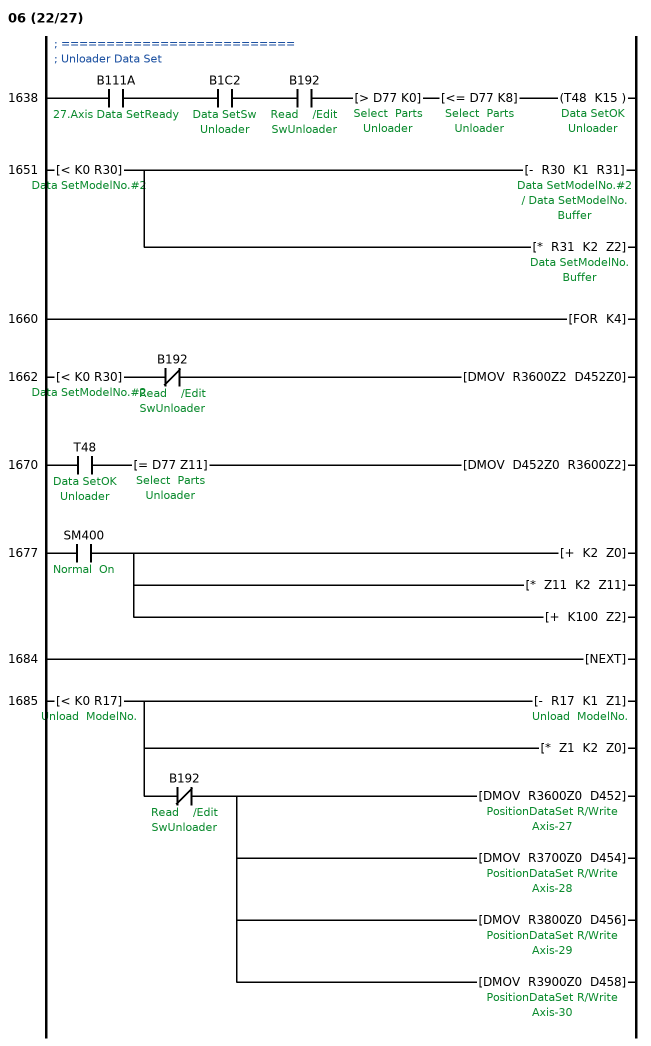
; ==========================
; Unloader Data Set
1638  LD      B111A  ; 27.Axis Data SetReady
      AND     B1C2  ; Data SetSw      Unloader
      AND     B192  ; Read    /Edit SwUnloader
      AND>    D77 K0  ; Select  Parts   Unloader
      AND<=   D77 K8  ; Select  Parts   Unloader
      OUT     T48 K15  ; Data SetOK      Unloader
1651  LD<     K0 R30  ; Data SetModelNo.#2
      -       R30 K1 R31
      *       R31 K2 Z2
1660  FOR     K4
1662  LD<     K0 R30  ; Data SetModelNo.#2
      ANI     B192  ; Read    /Edit SwUnloader
      DMOV    R3600Z2 D452Z0
1670  LD      T48  ; Data SetOK      Unloader
      AND=    D77 Z11  ; Select  Parts   Unloader
      DMOV    D452Z0 R3600Z2
1677  LD      SM400  ; Normal  On
      +       K2 Z0
      *       Z11 K2 Z11
      +       K100 Z2
1684  NEXT
1685  LD<     K0 R17  ; Unload  ModelNo.
      -       R17 K1 Z1
      *       Z1 K2 Z0
      ANI     B192  ; Read    /Edit SwUnloader
      DMOV    R3600Z0 D452  ; PositionDataSet R/Write Axis-27
      DMOV    R3700Z0 D454  ; PositionDataSet R/Write Axis-28
      DMOV    R3800Z0 D456  ; PositionDataSet R/Write Axis-29
      DMOV    R3900Z0 D458  ; PositionDataSet R/Write Axis-30
      P1
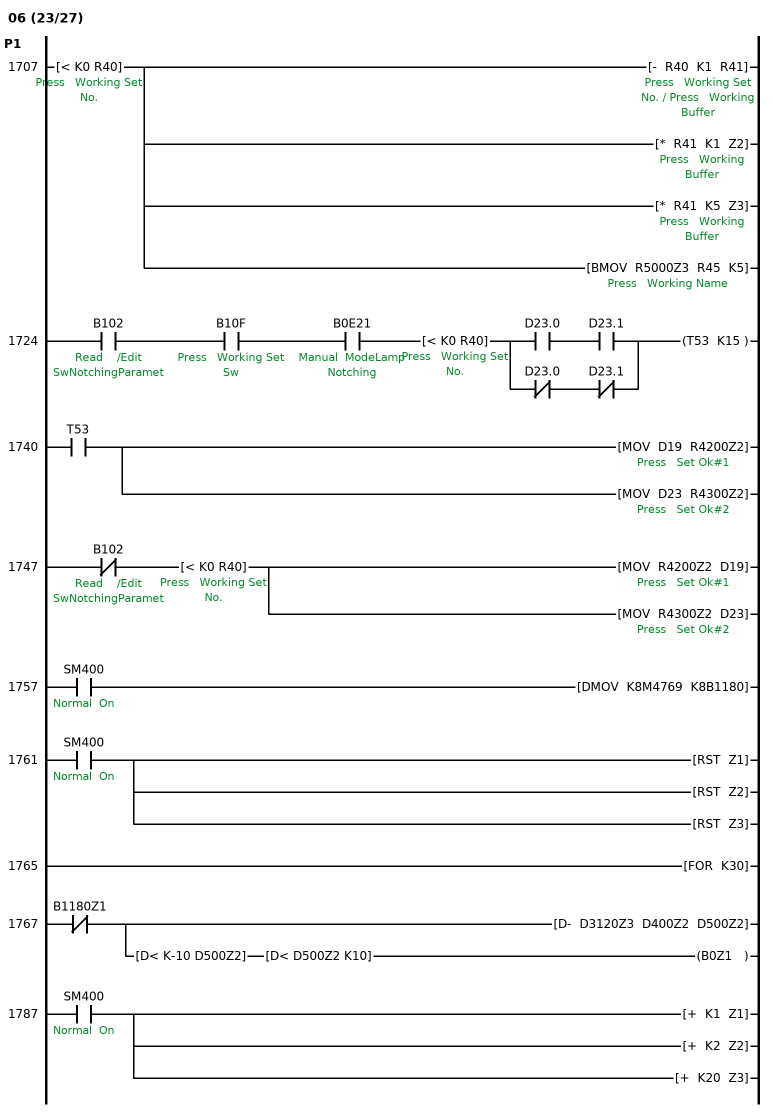
1707  LD<     K0 R40  ; Press   Working Set No.
      -       R40 K1 R41  ; Press   Working Buffer
      *       R41 K1 Z2
      *       R41 K5 Z3
      BMOV    R5000Z3 R45 K5  ; Press   Working Name
1724  LD      B102  ; Read    /Edit SwNotchingParamet
      AND     B10F  ; Press   Working Set Sw
      AND     B0E21  ; Manual  ModeLampNotching
      AND<    K0 R40  ; Press   Working Set No.
      LD      D23.0
      AND     D23.1
      LDI     D23.0
      ANI     D23.1
      ORB
      ANB
      OUT     T53 K15
1740  LD      T53
      MOV     D19 R4200Z2
      MOV     D23 R4300Z2
1747  LDI     B102  ; Read    /Edit SwNotchingParamet
      AND<    K0 R40  ; Press   Working Set No.
      MOV     R4200Z2 D19
      MOV     R4300Z2 D23
1757  LD      SM400  ; Normal  On
      DMOV    K8M4769 K8B1180  ; 1.Axis  Busy
1761  LD      SM400  ; Normal  On
      RST     Z1
      RST     Z2
      RST     Z3
1765  FOR     K30
1767  LDI     B1180Z1
      D-      D3120Z3 D400Z2 D500Z2
      ANDD<   K-10 D500Z2
      ANDD<   D500Z2 K10
      OUT     B0Z1
1787  LD      SM400  ; Normal  On
      +       K1 Z1
      +       K2 Z2
      +       K20 Z3
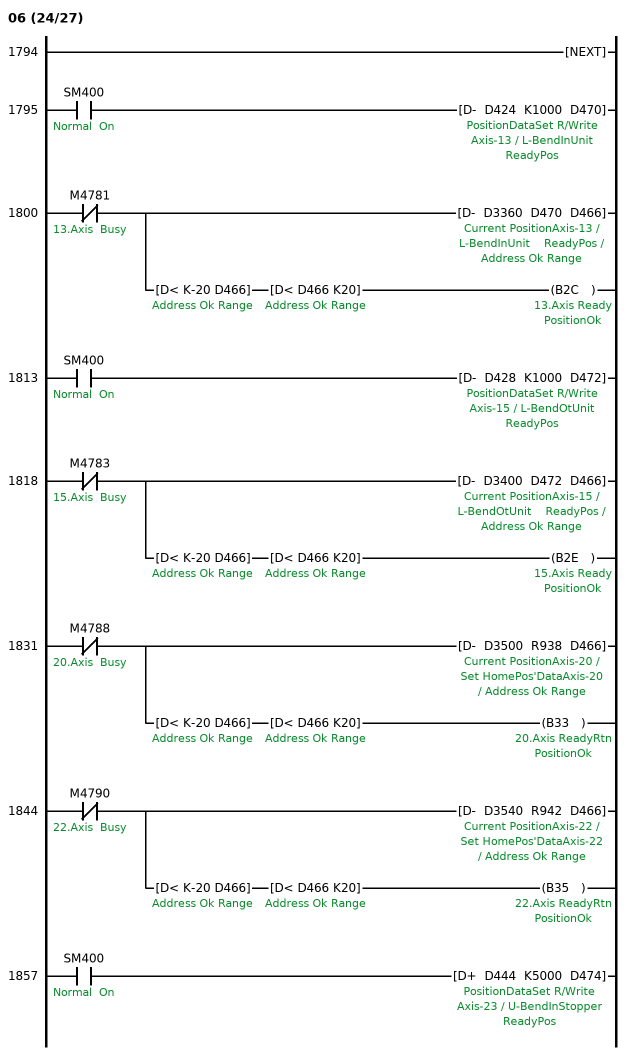
1794  NEXT
1795  LD      SM400  ; Normal  On
      D-      D424 K1000 D470  ; L-BendInUnit    ReadyPos
1800  LDI     M4781  ; 13.Axis  Busy
      D-      D3360 D470 D466  ; Current PositionAxis-13 / Address Ok Range
      ANDD<   K-20 D466  ; Address Ok Range
      ANDD<   D466 K20  ; Address Ok Range
      OUT     B2C  ; 13.Axis Ready   PositionOk
1813  LD      SM400  ; Normal  On
      D-      D428 K1000 D472  ; L-BendOtUnit    ReadyPos
1818  LDI     M4783  ; 15.Axis  Busy
      D-      D3400 D472 D466  ; Current PositionAxis-15
      ANDD<   K-20 D466  ; Address Ok Range
      ANDD<   D466 K20  ; Address Ok Range
      OUT     B2E  ; 15.Axis Ready   PositionOk
1831  LDI     M4788  ; 20.Axis  Busy
      D-      D3500 R938 D466  ; Current PositionAxis-20 / Set HomePos'DataAxis-20
      ANDD<   K-20 D466  ; Address Ok Range
      ANDD<   D466 K20  ; Address Ok Range
      OUT     B33  ; 20.Axis ReadyRtnPositionOk
1844  LDI     M4790  ; 22.Axis  Busy
      D-      D3540 R942 D466  ; Current PositionAxis-22 / Set HomePos'DataAxis-22
      ANDD<   K-20 D466  ; Address Ok Range
      ANDD<   D466 K20  ; Address Ok Range
      OUT     B35  ; 22.Axis ReadyRtnPositionOk
1857  LD      SM400  ; Normal  On
      D+      D444 K5000 D474  ; U-BendInStopper ReadyPos
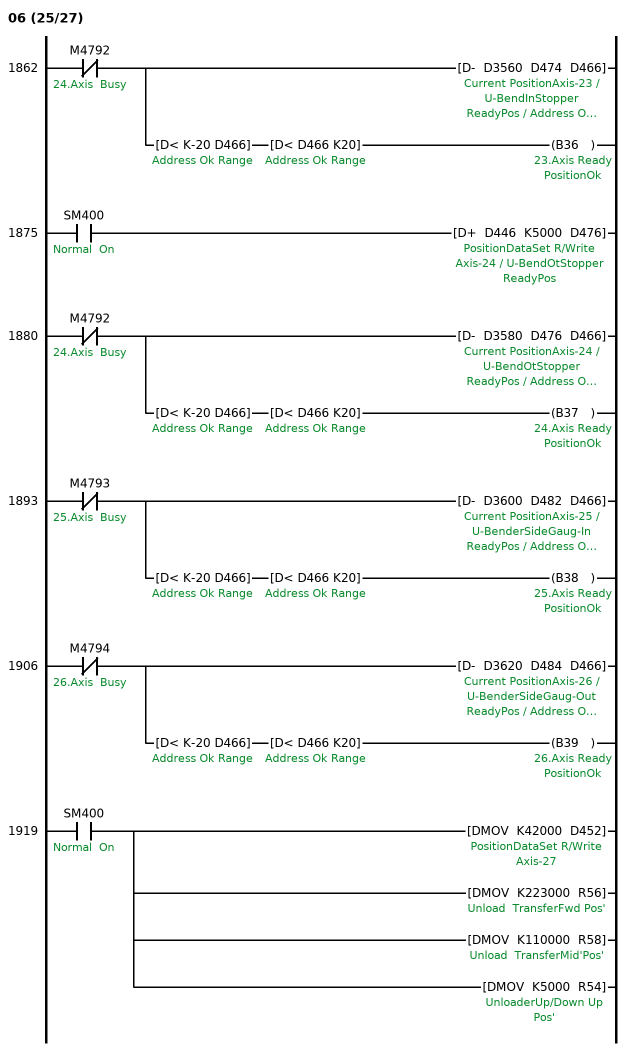
1862  LDI     M4792  ; 24.Axis  Busy
      D-      D3560 D474 D466  ; Current PositionAxis-23
      ANDD<   K-20 D466  ; Address Ok Range
      ANDD<   D466 K20  ; Address Ok Range
      OUT     B36  ; 23.Axis Ready   PositionOk
1875  LD      SM400  ; Normal  On
      D+      D446 K5000 D476  ; U-BendOtStopper ReadyPos
1880  LDI     M4792  ; 24.Axis  Busy
      D-      D3580 D476 D466  ; Current PositionAxis-24
      ANDD<   K-20 D466  ; Address Ok Range
      ANDD<   D466 K20  ; Address Ok Range
      OUT     B37  ; 24.Axis Ready   PositionOk
1893  LDI     M4793  ; 25.Axis  Busy
      D-      D3600 D482 D466  ; Current PositionAxis-25 / U-BenderSideGaug-In     ReadyPos
      ANDD<   K-20 D466  ; Address Ok Range
      ANDD<   D466 K20  ; Address Ok Range
      OUT     B38  ; 25.Axis Ready   PositionOk
1906  LDI     M4794  ; 26.Axis  Busy
      D-      D3620 D484 D466  ; Current PositionAxis-26 / U-BenderSideGaug-Out    ReadyPos
      ANDD<   K-20 D466  ; Address Ok Range
      ANDD<   D466 K20  ; Address Ok Range
      OUT     B39  ; 26.Axis Ready   PositionOk
1919  LD      SM400  ; Normal  On
      DMOV    K42000 D452
      DMOV    K223000 R56  ; Unload  TransferFwd Pos'
      DMOV    K110000 R58  ; Unload  TransferMid'Pos'
      DMOV    K5000 R54  ; UnloaderUp/Down Up Pos'
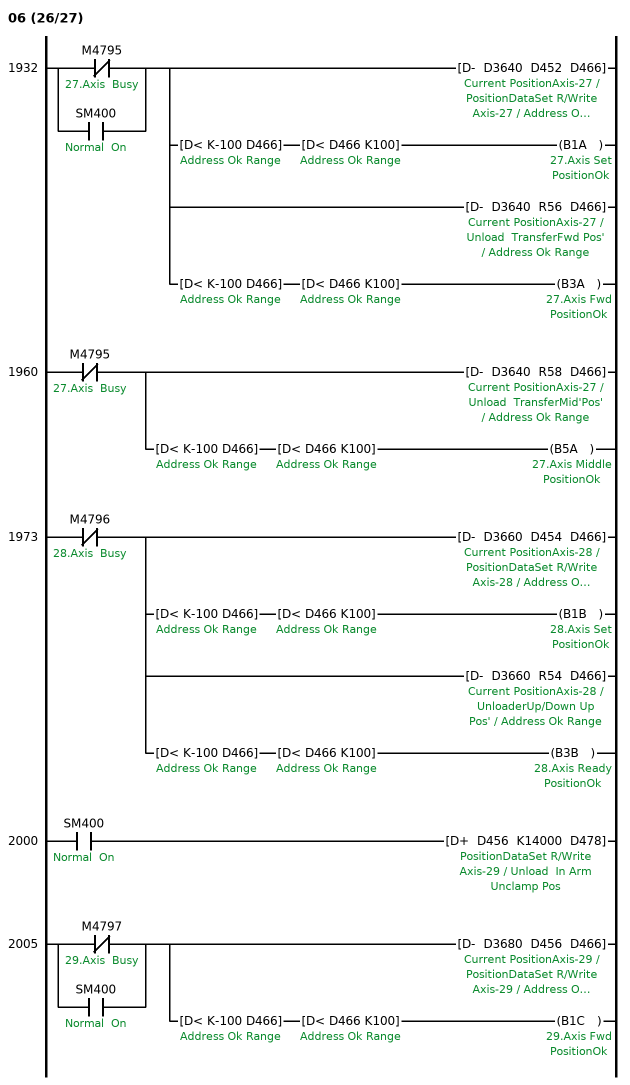
1932  LDI     M4795  ; 27.Axis  Busy
      OR      SM400  ; Normal  On
      D-      D3640 D452 D466  ; Current PositionAxis-27
      MPS
      ANDD<   K-100 D466  ; Address Ok Range
      ANDD<   D466 K100  ; Address Ok Range
      OUT     B1A  ; 27.Axis Set     PositionOk
      MPP
      D-      D3640 R56 D466
      ANDD<   K-100 D466  ; Address Ok Range
      ANDD<   D466 K100  ; Address Ok Range
      OUT     B3A  ; 27.Axis Fwd     PositionOk
1960  LDI     M4795  ; 27.Axis  Busy
      D-      D3640 R58 D466
      ANDD<   K-100 D466  ; Address Ok Range
      ANDD<   D466 K100  ; Address Ok Range
      OUT     B5A  ; 27.Axis Middle  PositionOk
1973  LDI     M4796  ; 28.Axis  Busy
      D-      D3660 D454 D466  ; Current PositionAxis-28
      MPS
      ANDD<   K-100 D466  ; Address Ok Range
      ANDD<   D466 K100  ; Address Ok Range
      OUT     B1B  ; 28.Axis Set     PositionOk
      MPP
      D-      D3660 R54 D466
      ANDD<   K-100 D466  ; Address Ok Range
      ANDD<   D466 K100  ; Address Ok Range
      OUT     B3B  ; 28.Axis Ready   PositionOk
2000  LD      SM400  ; Normal  On
      D+      D456 K14000 D478  ; Unload  In Arm  Unclamp Pos
2005  LDI     M4797  ; 29.Axis  Busy
      OR      SM400  ; Normal  On
      D-      D3680 D456 D466  ; Current PositionAxis-29
      ANDD<   K-100 D466  ; Address Ok Range
      ANDD<   D466 K100  ; Address Ok Range
      OUT     B1C  ; 29.Axis Fwd     PositionOk
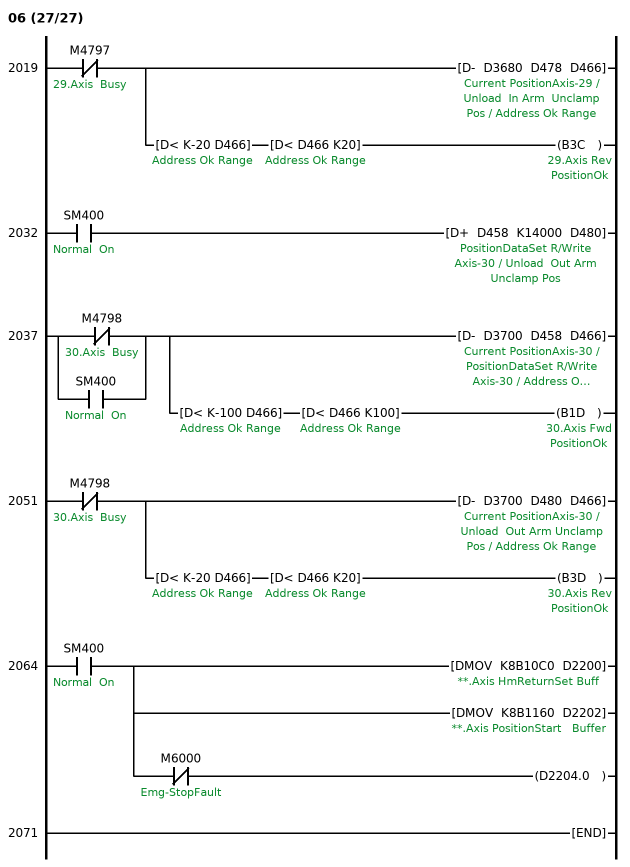
2019  LDI     M4797  ; 29.Axis  Busy
      D-      D3680 D478 D466
      ANDD<   K-20 D466  ; Address Ok Range
      ANDD<   D466 K20  ; Address Ok Range
      OUT     B3C  ; 29.Axis Rev     PositionOk
2032  LD      SM400  ; Normal  On
      D+      D458 K14000 D480  ; Unload  Out Arm Unclamp Pos
2037  LDI     M4798  ; 30.Axis  Busy
      OR      SM400  ; Normal  On
      D-      D3700 D458 D466  ; Current PositionAxis-30
      ANDD<   K-100 D466  ; Address Ok Range
      ANDD<   D466 K100  ; Address Ok Range
      OUT     B1D  ; 30.Axis Fwd     PositionOk
2051  LDI     M4798  ; 30.Axis  Busy
      D-      D3700 D480 D466
      ANDD<   K-20 D466  ; Address Ok Range
      ANDD<   D466 K20  ; Address Ok Range
      OUT     B3D  ; 30.Axis Rev     PositionOk
2064  LD      SM400  ; Normal  On
      DMOV    K8B10C0 D2200  ; 01.Axis HmReturnSet / **.Axis HmReturnSet Buff
      DMOV    K8B1160 D2202  ; 01.Axis PositionStart / **.Axis PositionStart   Buffer
      ANI     M6000  ; Emg-StopFault
      OUT     D2204.0
2071  END
END_PROGRAM

PROGRAM 10  // #1 Conveyor Part
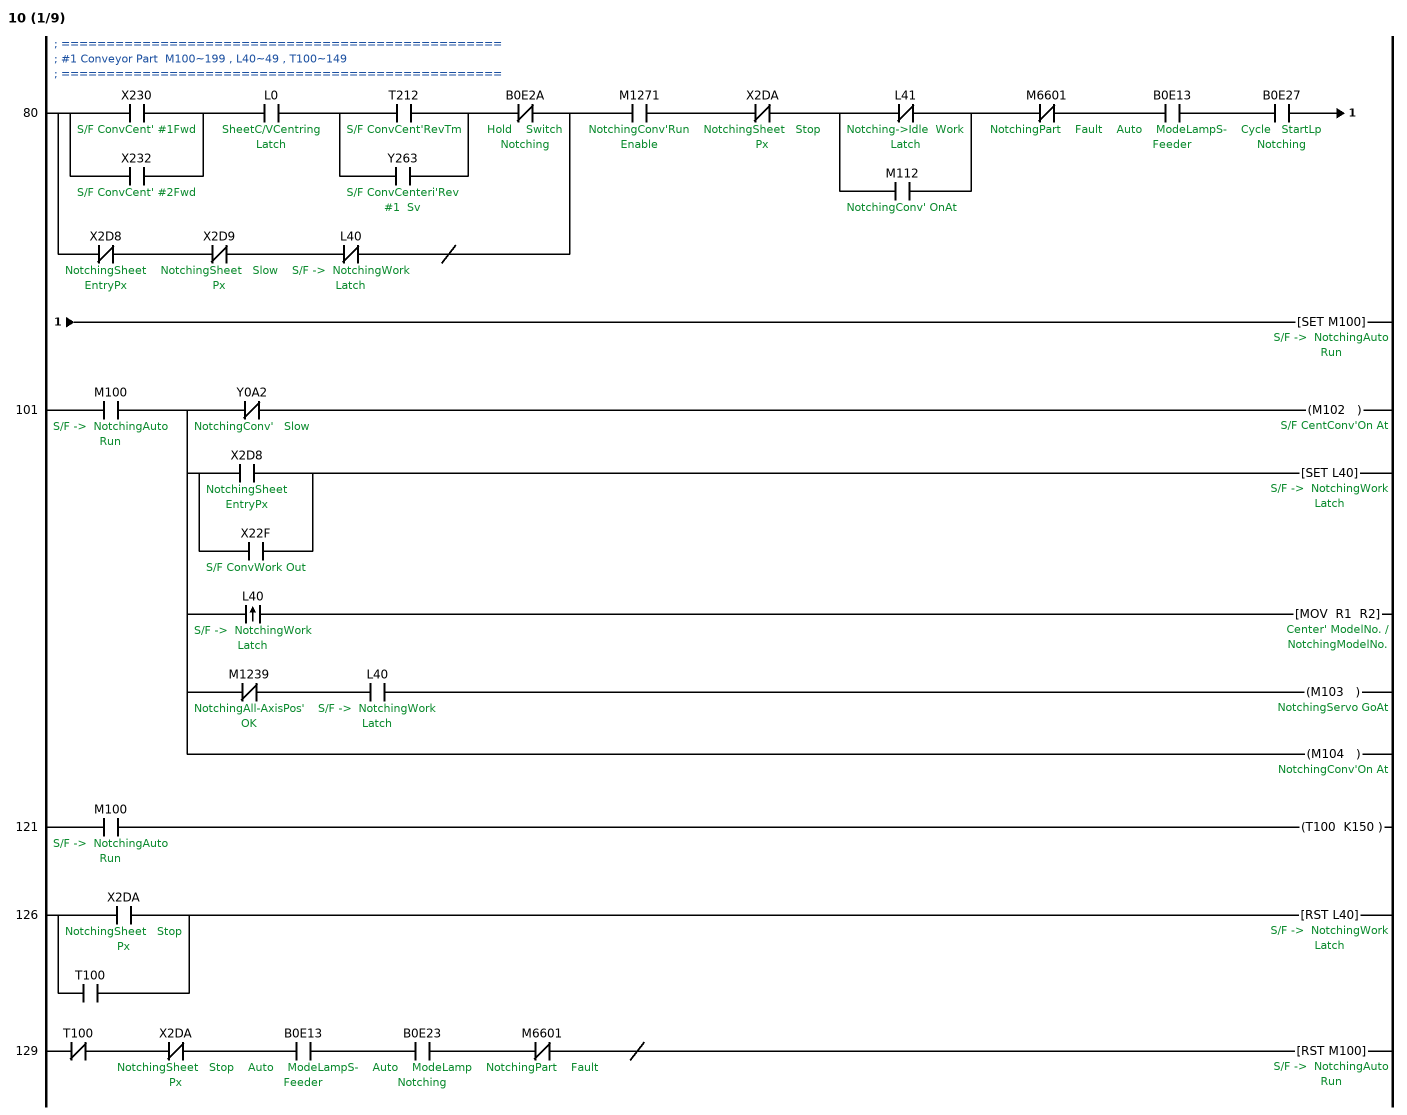
; =================================================
; #1 Conveyor Part  M100~199 , L40~49 , T100~149
; =================================================
80    LD      X230  ; S/F ConvCent' #1Fwd
      OR      X232  ; S/F ConvCent' #2Fwd
      AND     L0  ; SheetC/VCentringLatch
      LD      T212  ; S/F ConvCent'RevTm
      OR      Y263  ; S/F ConvCenteri'Rev #1  Sv
      ANB
      ANI     B0E2A  ; Hold    Switch  Notching
      LDI     X2D8  ; NotchingSheet   EntryPx
      ANI     X2D9  ; NotchingSheet   Slow Px
      ANI     L40  ; S/F ->  NotchingWork    Latch
      INV
      ORB
      AND     M1271  ; NotchingConv'RunEnable
      ANI     X2DA  ; NotchingSheet   Stop Px
      LDI     L41  ; Notching->Idle  Work    Latch
      OR      M112  ; NotchingConv' OnAt
      ANB
      ANI     M6601  ; NotchingPart    Fault
      AND     B0E13  ; Auto    ModeLampS-Feeder
      AND     B0E27  ; Cycle   StartLp Notching
      SET     M100  ; S/F ->  NotchingAuto Run
101   LD      M100  ; S/F ->  NotchingAuto Run
      MPS
      ANI     Y0A2  ; NotchingConv'   Slow
      OUT     M102  ; S/F CentConv'On At
      MRD
      LD      X2D8  ; NotchingSheet   EntryPx
      OR      X22F  ; S/F ConvWork Out
      ANB
      SET     L40  ; S/F ->  NotchingWork    Latch
      MRD
      ANDP    L40  ; S/F ->  NotchingWork    Latch
      MOV     R1 R2  ; Center' ModelNo. / NotchingModelNo.
      MRD
      ANI     M1239  ; NotchingAll-AxisPos' OK
      AND     L40  ; S/F ->  NotchingWork    Latch
      OUT     M103  ; NotchingServo GoAt
      MPP
      OUT     M104  ; NotchingConv'On At
121   LD      M100  ; S/F ->  NotchingAuto Run
      OUT     T100 K150
126   LD      X2DA  ; NotchingSheet   Stop Px
      OR      T100
      RST     L40  ; S/F ->  NotchingWork    Latch
129   LDI     T100
      ANI     X2DA  ; NotchingSheet   Stop Px
      AND     B0E13  ; Auto    ModeLampS-Feeder
      AND     B0E23  ; Auto    ModeLampNotching
      ANI     M6601  ; NotchingPart    Fault
      INV
      RST     M100  ; S/F ->  NotchingAuto Run
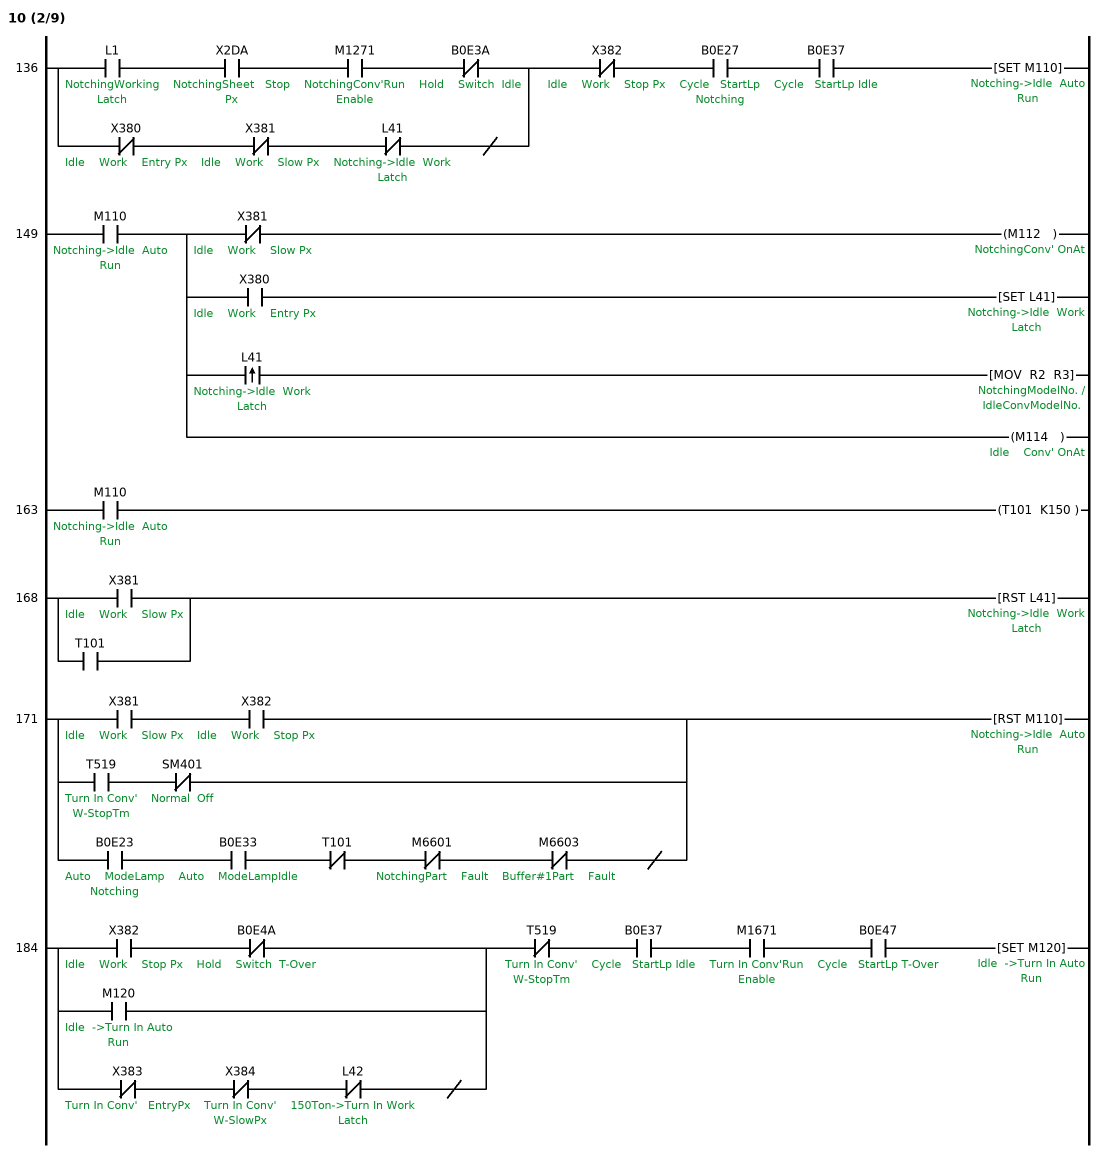
136   LD      L1  ; NotchingWorking Latch
      AND     X2DA  ; NotchingSheet   Stop Px
      AND     M1271  ; NotchingConv'RunEnable
      ANI     B0E3A  ; Hold    Switch  Idle
      LDI     X380  ; Idle    Work    Entry Px
      ANI     X381  ; Idle    Work    Slow Px
      ANI     L41  ; Notching->Idle  Work    Latch
      INV
      ORB
      ANI     X382  ; Idle    Work    Stop Px
      AND     B0E27  ; Cycle   StartLp Notching
      AND     B0E37  ; Cycle   StartLp Idle
      SET     M110  ; Notching->Idle  Auto Run
149   LD      M110  ; Notching->Idle  Auto Run
      MPS
      ANI     X381  ; Idle    Work    Slow Px
      OUT     M112  ; NotchingConv' OnAt
      MRD
      AND     X380  ; Idle    Work    Entry Px
      SET     L41  ; Notching->Idle  Work    Latch
      MRD
      ANDP    L41  ; Notching->Idle  Work    Latch
      MOV     R2 R3  ; IdleConvModelNo.
      MPP
      OUT     M114  ; Idle    Conv' OnAt
163   LD      M110  ; Notching->Idle  Auto Run
      OUT     T101 K150
168   LD      X381  ; Idle    Work    Slow Px
      OR      T101
      RST     L41  ; Notching->Idle  Work    Latch
171   LD      X381  ; Idle    Work    Slow Px
      AND     X382  ; Idle    Work    Stop Px
      LD      T519  ; Turn In Conv'   W-StopTm
      ANI     SM401  ; Normal  Off
      ORB
      LD      B0E23  ; Auto    ModeLampNotching
      AND     B0E33  ; Auto    ModeLampIdle
      ANI     T101
      ANI     M6601  ; NotchingPart    Fault
      ANI     M6603  ; Buffer#1Part    Fault
      INV
      ORB
      RST     M110  ; Notching->Idle  Auto Run
184   LD      X382  ; Idle    Work    Stop Px
      ANI     B0E4A  ; Hold    Switch  T-Over
      OR      M120  ; Idle  ->Turn In Auto Run
      LDI     X383  ; Turn In Conv'   EntryPx
      ANI     X384  ; Turn In Conv'   W-SlowPx
      ANI     L42  ; 150Ton->Turn In Work    Latch
      INV
      ORB
      ANI     T519  ; Turn In Conv'   W-StopTm
      AND     B0E37  ; Cycle   StartLp Idle
      AND     M1671  ; Turn In Conv'RunEnable
      AND     B0E47  ; Cycle   StartLp T-Over
      SET     M120  ; Idle  ->Turn In Auto Run
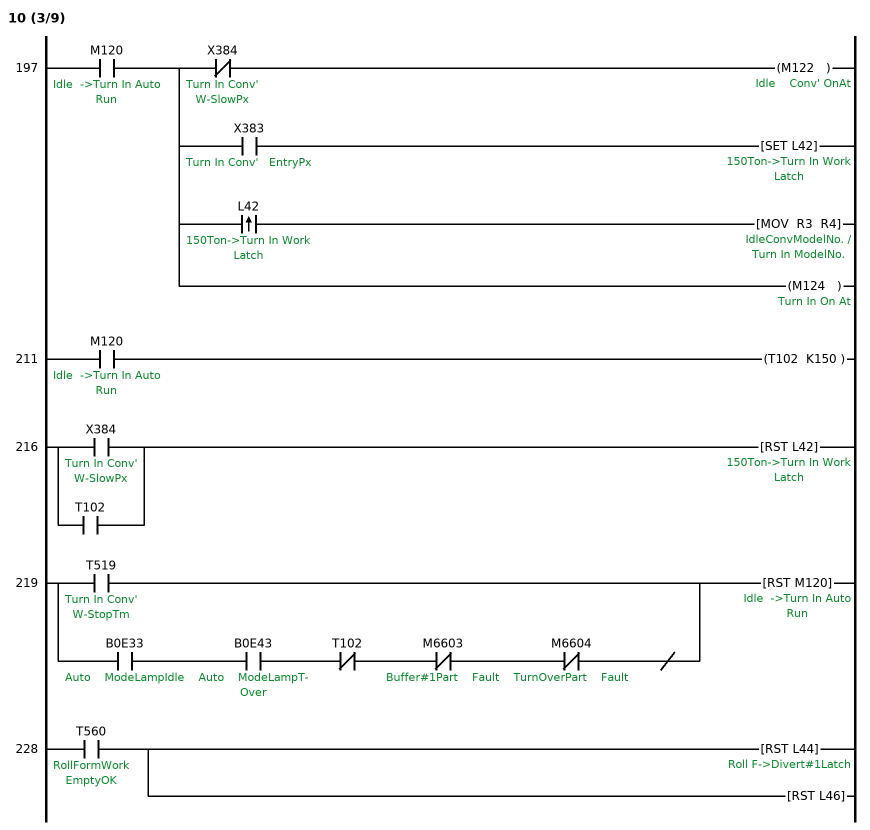
197   LD      M120  ; Idle  ->Turn In Auto Run
      MPS
      ANI     X384  ; Turn In Conv'   W-SlowPx
      OUT     M122  ; Idle    Conv' OnAt
      MRD
      AND     X383  ; Turn In Conv'   EntryPx
      SET     L42  ; 150Ton->Turn In Work    Latch
      MRD
      ANDP    L42  ; 150Ton->Turn In Work    Latch
      MOV     R3 R4  ; Turn In ModelNo.
      MPP
      OUT     M124  ; Turn In On At
211   LD      M120  ; Idle  ->Turn In Auto Run
      OUT     T102 K150
216   LD      X384  ; Turn In Conv'   W-SlowPx
      OR      T102
      RST     L42  ; 150Ton->Turn In Work    Latch
219   LD      T519  ; Turn In Conv'   W-StopTm
      LD      B0E33  ; Auto    ModeLampIdle
      AND     B0E43  ; Auto    ModeLampT-Over
      ANI     T102
      ANI     M6603  ; Buffer#1Part    Fault
      ANI     M6604  ; TurnOverPart    Fault
      INV
      ORB
      RST     M120  ; Idle  ->Turn In Auto Run
228   LD      T560  ; RollFormWork    EmptyOK
      RST     L44  ; Roll F->Divert#1Latch
      RST     L46
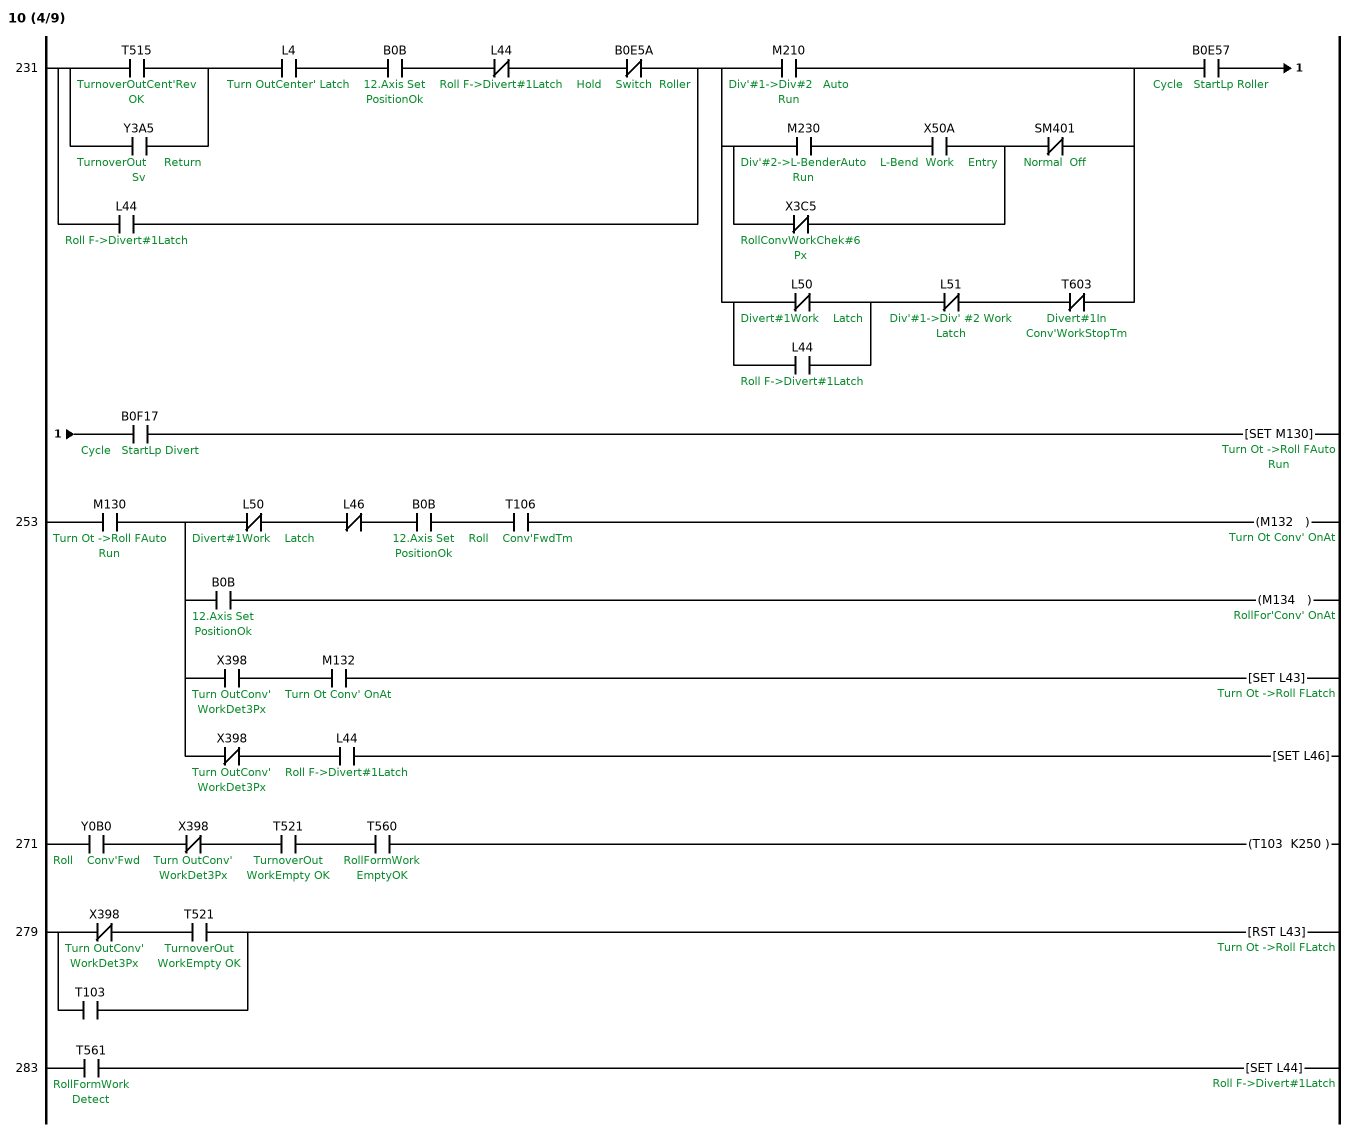
231   LD      T515  ; TurnoverOutCent'Rev OK
      OR      Y3A5  ; TurnoverOut     Return  Sv
      AND     L4  ; Turn OutCenter' Latch
      AND     B0B  ; 12.Axis Set     PositionOk
      ANI     L44  ; Roll F->Divert#1Latch
      ANI     B0E5A  ; Hold    Switch  Roller
      OR      L44  ; Roll F->Divert#1Latch
      LD      M210  ; Div'#1->Div#2   Auto Run
      LD      M230  ; Div'#2->L-BenderAuto Run
      AND     X50A  ; L-Bend  Work    Entry
      ORI     X3C5  ; RollConvWorkChek#6 Px
      ANI     SM401  ; Normal  Off
      ORB
      LDI     L50  ; Divert#1Work    Latch
      OR      L44  ; Roll F->Divert#1Latch
      ANI     L51  ; Div'#1->Div' #2 Work    Latch
      ANI     T603  ; Divert#1In Conv'WorkStopTm
      ORB
      ANB
      AND     B0E57  ; Cycle   StartLp Roller
      AND     B0F17  ; Cycle   StartLp Divert
      SET     M130  ; Turn Ot ->Roll FAuto Run
253   LD      M130  ; Turn Ot ->Roll FAuto Run
      MPS
      ANI     L50  ; Divert#1Work    Latch
      ANI     L46
      AND     B0B  ; 12.Axis Set     PositionOk
      AND     T106  ; Roll    Conv'FwdTm
      OUT     M132  ; Turn Ot Conv' OnAt
      MRD
      AND     B0B  ; 12.Axis Set     PositionOk
      OUT     M134  ; RollFor'Conv' OnAt
      MRD
      AND     X398  ; Turn OutConv'   WorkDet3Px
      AND     M132  ; Turn Ot Conv' OnAt
      SET     L43  ; Turn Ot ->Roll FLatch
      MPP
      ANI     X398  ; Turn OutConv'   WorkDet3Px
      AND     L44  ; Roll F->Divert#1Latch
      SET     L46
271   LD      Y0B0  ; Roll    Conv'Fwd
      ANI     X398  ; Turn OutConv'   WorkDet3Px
      AND     T521  ; TurnoverOut WorkEmpty OK
      AND     T560  ; RollFormWork    EmptyOK
      OUT     T103 K250
279   LDI     X398  ; Turn OutConv'   WorkDet3Px
      AND     T521  ; TurnoverOut WorkEmpty OK
      OR      T103
      RST     L43  ; Turn Ot ->Roll FLatch
283   LD      T561  ; RollFormWork    Detect
      SET     L44  ; Roll F->Divert#1Latch
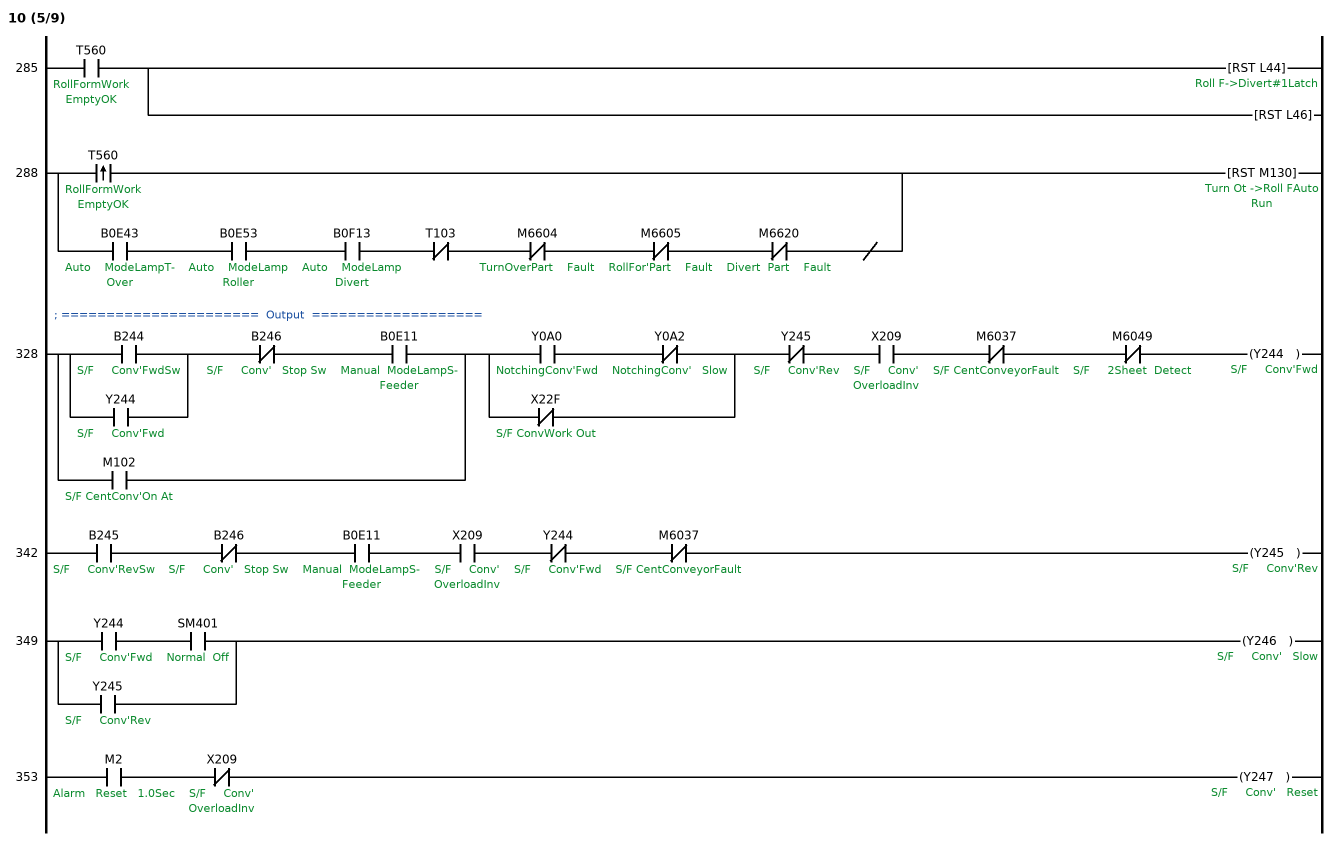
285   LD      T560  ; RollFormWork    EmptyOK
      RST     L44  ; Roll F->Divert#1Latch
      RST     L46
288   LDP     T560  ; RollFormWork    EmptyOK
      LD      B0E43  ; Auto    ModeLampT-Over
      AND     B0E53  ; Auto    ModeLampRoller
      AND     B0F13  ; Auto    ModeLampDivert
      ANI     T103
      ANI     M6604  ; TurnOverPart    Fault
      ANI     M6605  ; RollFor'Part    Fault
      ANI     M6620  ; Divert  Part    Fault
      INV
      ORB
      RST     M130  ; Turn Ot ->Roll FAuto Run
; ======================  Output  ===================
328   LD      B244  ; S/F     Conv'FwdSw
      OR      Y244  ; S/F     Conv'Fwd
      ANI     B246  ; S/F     Conv'   Stop Sw
      AND     B0E11  ; Manual  ModeLampS-Feeder
      OR      M102  ; S/F CentConv'On At
      LD      Y0A0  ; NotchingConv'Fwd
      ANI     Y0A2  ; NotchingConv'   Slow
      ORI     X22F  ; S/F ConvWork Out
      ANB
      ANI     Y245  ; S/F     Conv'Rev
      AND     X209  ; S/F     Conv'   OverloadInv
      ANI     M6037  ; S/F CentConveyorFault
      ANI     M6049  ; S/F     2Sheet  Detect
      OUT     Y244  ; S/F     Conv'Fwd
342   LD      B245  ; S/F     Conv'RevSw
      ANI     B246  ; S/F     Conv'   Stop Sw
      AND     B0E11  ; Manual  ModeLampS-Feeder
      AND     X209  ; S/F     Conv'   OverloadInv
      ANI     Y244  ; S/F     Conv'Fwd
      ANI     M6037  ; S/F CentConveyorFault
      OUT     Y245  ; S/F     Conv'Rev
349   LD      Y244  ; S/F     Conv'Fwd
      AND     SM401  ; Normal  Off
      OR      Y245  ; S/F     Conv'Rev
      OUT     Y246  ; S/F     Conv'   Slow
353   LD      M2  ; Alarm   Reset   1.0Sec
      ANI     X209  ; S/F     Conv'   OverloadInv
      OUT     Y247  ; S/F     Conv'   Reset
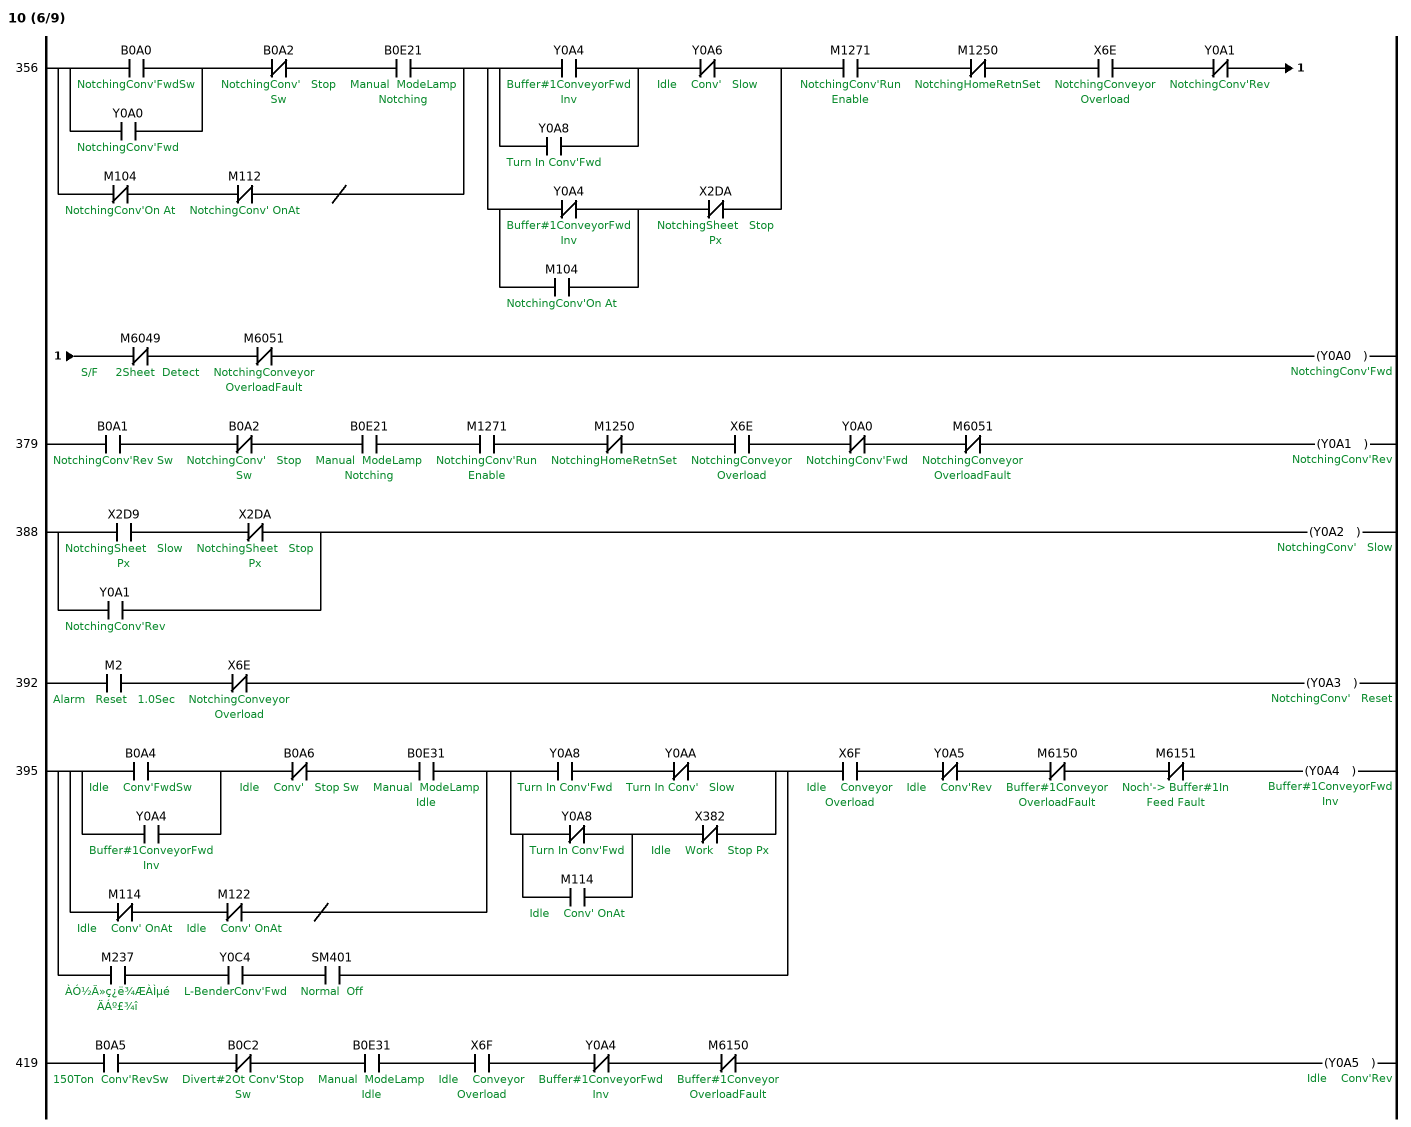
356   LD      B0A0  ; NotchingConv'FwdSw
      OR      Y0A0  ; NotchingConv'Fwd
      ANI     B0A2  ; NotchingConv'   Stop Sw
      AND     B0E21  ; Manual  ModeLampNotching
      LDI     M104  ; NotchingConv'On At
      ANI     M112  ; NotchingConv' OnAt
      INV
      ORB
      LD      Y0A4  ; Buffer#1ConveyorFwd Inv
      OR      Y0A8  ; Turn In Conv'Fwd
      ANI     Y0A6  ; Idle    Conv'   Slow
      LDI     Y0A4  ; Buffer#1ConveyorFwd Inv
      OR      M104  ; NotchingConv'On At
      ANI     X2DA  ; NotchingSheet   Stop Px
      ORB
      ANB
      AND     M1271  ; NotchingConv'RunEnable
      ANI     M1250  ; NotchingHomeRetnSet
      AND     X6E  ; NotchingConveyorOverload
      ANI     Y0A1  ; NotchingConv'Rev
      ANI     M6049  ; S/F     2Sheet  Detect
      ANI     M6051  ; NotchingConveyorOverloadFault
      OUT     Y0A0  ; NotchingConv'Fwd
379   LD      B0A1  ; NotchingConv'Rev Sw
      ANI     B0A2  ; NotchingConv'   Stop Sw
      AND     B0E21  ; Manual  ModeLampNotching
      AND     M1271  ; NotchingConv'RunEnable
      ANI     M1250  ; NotchingHomeRetnSet
      AND     X6E  ; NotchingConveyorOverload
      ANI     Y0A0  ; NotchingConv'Fwd
      ANI     M6051  ; NotchingConveyorOverloadFault
      OUT     Y0A1  ; NotchingConv'Rev
388   LD      X2D9  ; NotchingSheet   Slow Px
      ANI     X2DA  ; NotchingSheet   Stop Px
      OR      Y0A1  ; NotchingConv'Rev
      OUT     Y0A2  ; NotchingConv'   Slow
392   LD      M2  ; Alarm   Reset   1.0Sec
      ANI     X6E  ; NotchingConveyorOverload
      OUT     Y0A3  ; NotchingConv'   Reset
395   LD      B0A4  ; Idle    Conv'FwdSw
      OR      Y0A4  ; Buffer#1ConveyorFwd Inv
      ANI     B0A6  ; Idle    Conv'   Stop Sw
      AND     B0E31  ; Manual  ModeLampIdle
      LDI     M114  ; Idle    Conv' OnAt
      ANI     M122  ; Idle    Conv' OnAt
      INV
      ORB
      LD      Y0A8  ; Turn In Conv'Fwd
      ANI     Y0AA  ; Turn In Conv'   Slow
      LDI     Y0A8  ; Turn In Conv'Fwd
      OR      M114  ; Idle    Conv' OnAt
      ANI     X382  ; Idle    Work    Stop Px
      ORB
      ANB
      LD      M237  ; ÀÓ½Ã»ç¿ë¾ÆÀÌµéÄÁº£¾î
      AND     Y0C4  ; L-BenderConv'Fwd
      AND     SM401  ; Normal  Off
      ORB
      AND     X6F  ; Idle    ConveyorOverload
      ANI     Y0A5  ; Idle    Conv'Rev
      ANI     M6150  ; Buffer#1ConveyorOverloadFault
      ANI     M6151  ; Noch'-> Buffer#1In Feed Fault
      OUT     Y0A4  ; Buffer#1ConveyorFwd Inv
419   LD      B0A5  ; 150Ton  Conv'RevSw
      ANI     B0C2  ; Divert#2Ot Conv'Stop Sw
      AND     B0E31  ; Manual  ModeLampIdle
      AND     X6F  ; Idle    ConveyorOverload
      ANI     Y0A4  ; Buffer#1ConveyorFwd Inv
      ANI     M6150  ; Buffer#1ConveyorOverloadFault
      OUT     Y0A5  ; Idle    Conv'Rev
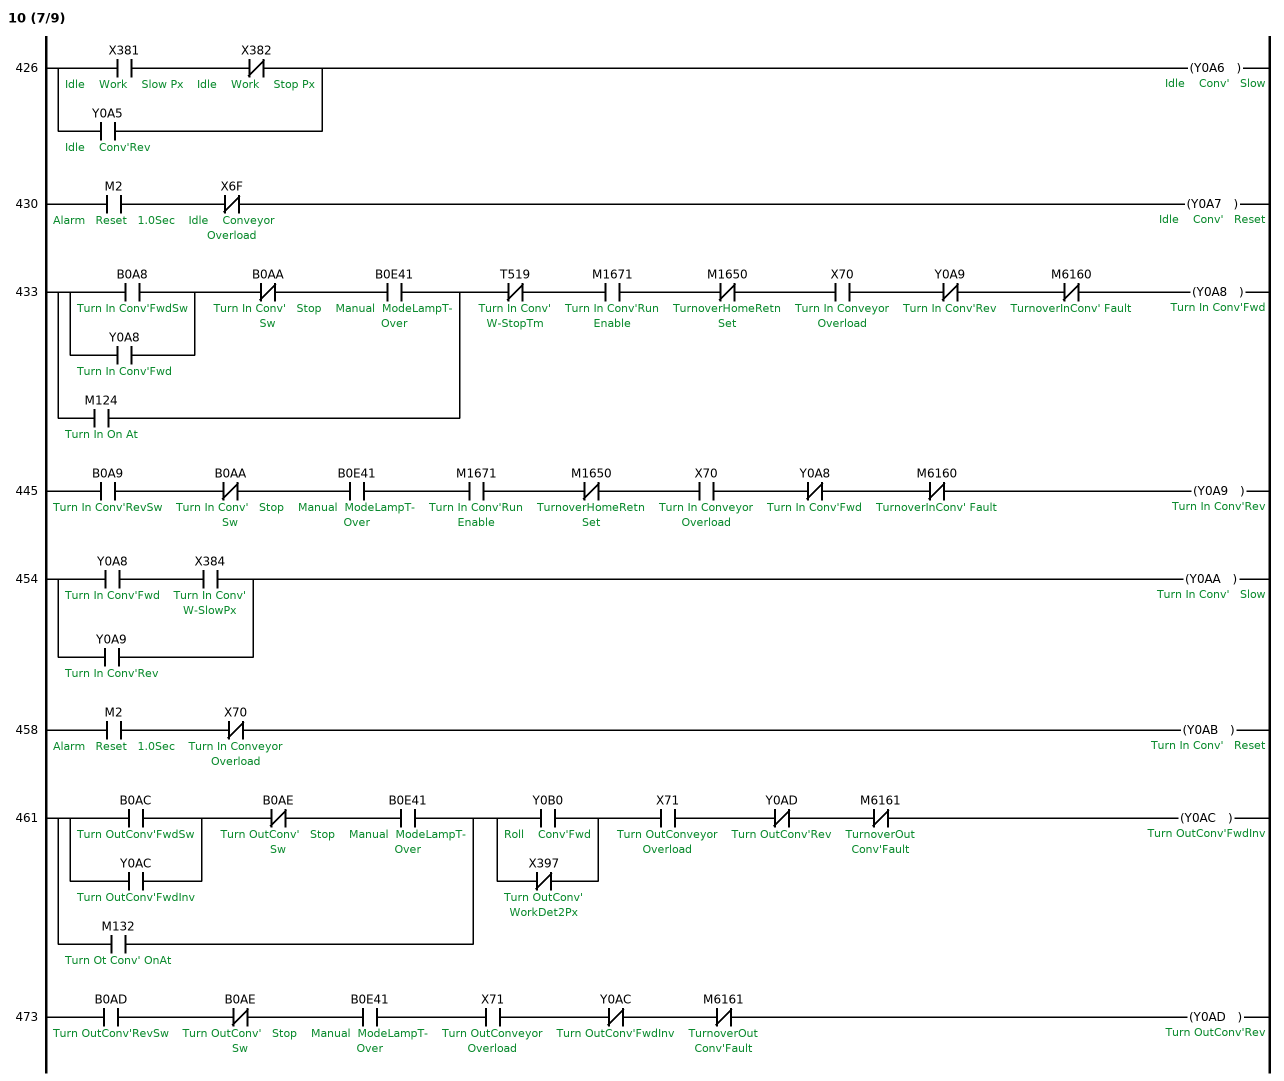
426   LD      X381  ; Idle    Work    Slow Px
      ANI     X382  ; Idle    Work    Stop Px
      OR      Y0A5  ; Idle    Conv'Rev
      OUT     Y0A6  ; Idle    Conv'   Slow
430   LD      M2  ; Alarm   Reset   1.0Sec
      ANI     X6F  ; Idle    ConveyorOverload
      OUT     Y0A7  ; Idle    Conv'   Reset
433   LD      B0A8  ; Turn In Conv'FwdSw
      OR      Y0A8  ; Turn In Conv'Fwd
      ANI     B0AA  ; Turn In Conv'   Stop Sw
      AND     B0E41  ; Manual  ModeLampT-Over
      OR      M124  ; Turn In On At
      ANI     T519  ; Turn In Conv'   W-StopTm
      AND     M1671  ; Turn In Conv'RunEnable
      ANI     M1650  ; TurnoverHomeRetnSet
      AND     X70  ; Turn In ConveyorOverload
      ANI     Y0A9  ; Turn In Conv'Rev
      ANI     M6160  ; TurnoverInConv' Fault
      OUT     Y0A8  ; Turn In Conv'Fwd
445   LD      B0A9  ; Turn In Conv'RevSw
      ANI     B0AA  ; Turn In Conv'   Stop Sw
      AND     B0E41  ; Manual  ModeLampT-Over
      AND     M1671  ; Turn In Conv'RunEnable
      ANI     M1650  ; TurnoverHomeRetnSet
      AND     X70  ; Turn In ConveyorOverload
      ANI     Y0A8  ; Turn In Conv'Fwd
      ANI     M6160  ; TurnoverInConv' Fault
      OUT     Y0A9  ; Turn In Conv'Rev
454   LD      Y0A8  ; Turn In Conv'Fwd
      AND     X384  ; Turn In Conv'   W-SlowPx
      OR      Y0A9  ; Turn In Conv'Rev
      OUT     Y0AA  ; Turn In Conv'   Slow
458   LD      M2  ; Alarm   Reset   1.0Sec
      ANI     X70  ; Turn In ConveyorOverload
      OUT     Y0AB  ; Turn In Conv'   Reset
461   LD      B0AC  ; Turn OutConv'FwdSw
      OR      Y0AC  ; Turn OutConv'FwdInv
      ANI     B0AE  ; Turn OutConv'   Stop Sw
      AND     B0E41  ; Manual  ModeLampT-Over
      OR      M132  ; Turn Ot Conv' OnAt
      LD      Y0B0  ; Roll    Conv'Fwd
      ORI     X397  ; Turn OutConv'   WorkDet2Px
      ANB
      AND     X71  ; Turn OutConveyorOverload
      ANI     Y0AD  ; Turn OutConv'Rev
      ANI     M6161  ; TurnoverOutConv'Fault
      OUT     Y0AC  ; Turn OutConv'FwdInv
473   LD      B0AD  ; Turn OutConv'RevSw
      ANI     B0AE  ; Turn OutConv'   Stop Sw
      AND     B0E41  ; Manual  ModeLampT-Over
      AND     X71  ; Turn OutConveyorOverload
      ANI     Y0AC  ; Turn OutConv'FwdInv
      ANI     M6161  ; TurnoverOutConv'Fault
      OUT     Y0AD  ; Turn OutConv'Rev
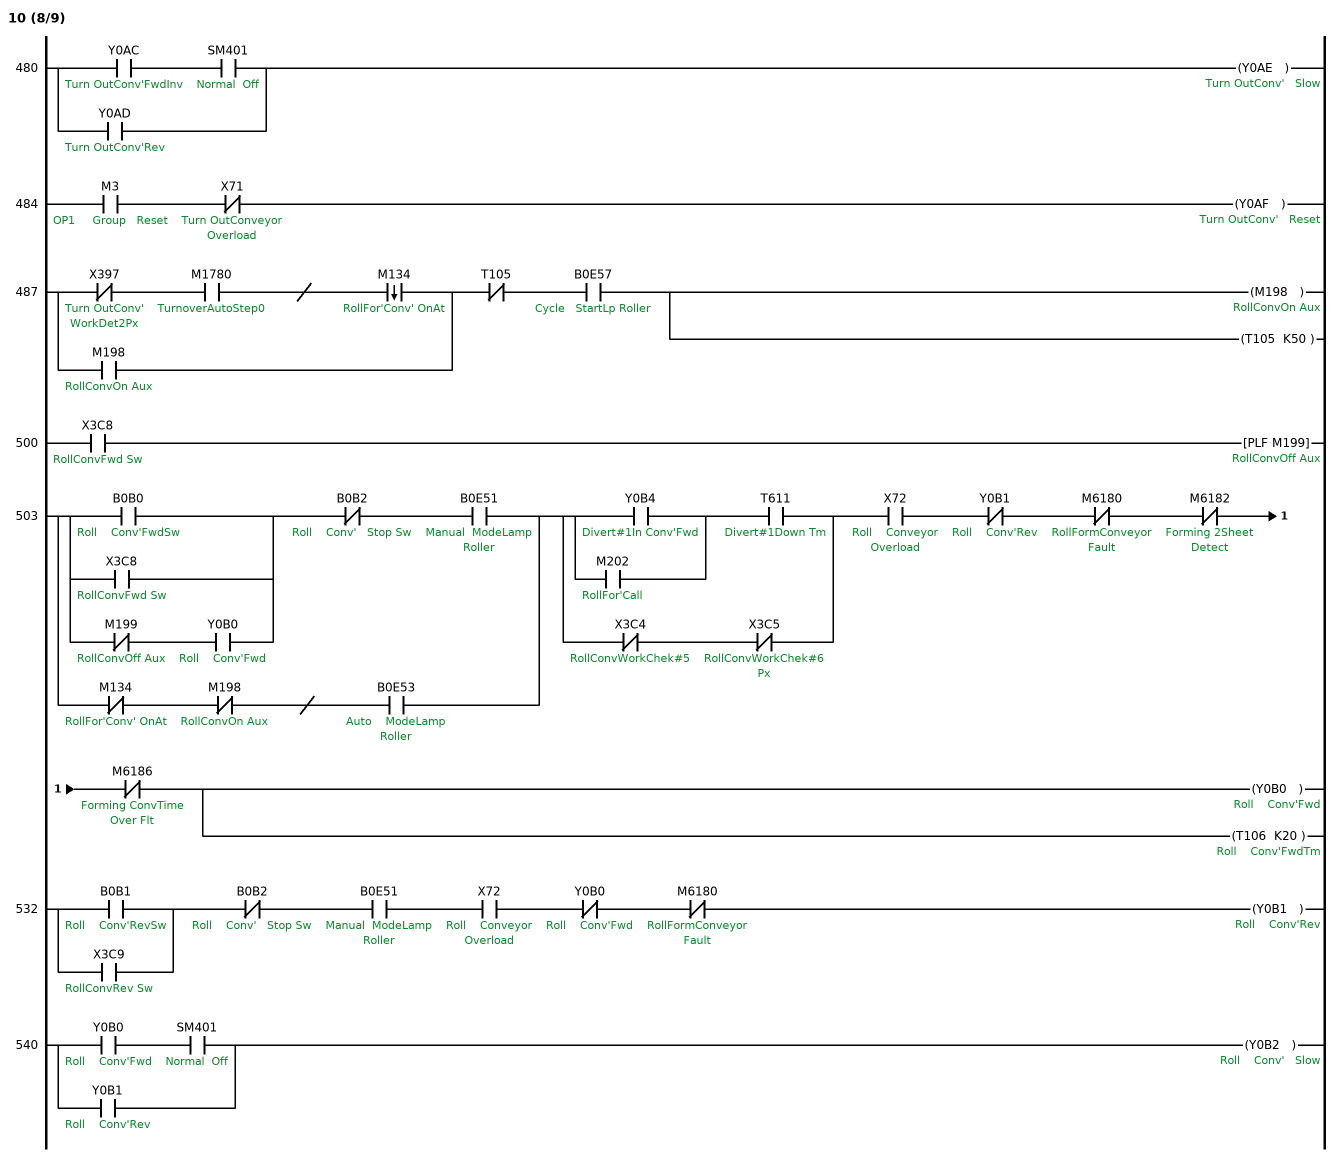
480   LD      Y0AC  ; Turn OutConv'FwdInv
      AND     SM401  ; Normal  Off
      OR      Y0AD  ; Turn OutConv'Rev
      OUT     Y0AE  ; Turn OutConv'   Slow
484   LD      M3  ; OP1     Group   Reset
      ANI     X71  ; Turn OutConveyorOverload
      OUT     Y0AF  ; Turn OutConv'   Reset
487   LDI     X397  ; Turn OutConv'   WorkDet2Px
      AND     M1780  ; TurnoverAutoStep0
      INV
      ANDF    M134  ; RollFor'Conv' OnAt
      OR      M198  ; RollConvOn Aux
      ANI     T105
      AND     B0E57  ; Cycle   StartLp Roller
      OUT     M198  ; RollConvOn Aux
      OUT     T105 K50
500   LD      X3C8  ; RollConvFwd Sw
      PLF     M199  ; RollConvOff Aux
503   LD      B0B0  ; Roll    Conv'FwdSw
      OR      X3C8  ; RollConvFwd Sw
      LDI     M199  ; RollConvOff Aux
      AND     Y0B0  ; Roll    Conv'Fwd
      ORB
      ANI     B0B2  ; Roll    Conv'   Stop Sw
      AND     B0E51  ; Manual  ModeLampRoller
      LDI     M134  ; RollFor'Conv' OnAt
      ANI     M198  ; RollConvOn Aux
      INV
      AND     B0E53  ; Auto    ModeLampRoller
      ORB
      LD      Y0B4  ; Divert#1In Conv'Fwd
      OR      M202  ; RollFor'Call
      AND     T611  ; Divert#1Down Tm
      LDI     X3C4  ; RollConvWorkChek#5
      ANI     X3C5  ; RollConvWorkChek#6 Px
      ORB
      ANB
      AND     X72  ; Roll    ConveyorOverload
      ANI     Y0B1  ; Roll    Conv'Rev
      ANI     M6180  ; RollFormConveyorFault
      ANI     M6182  ; Forming 2Sheet  Detect
      ANI     M6186  ; Forming ConvTimeOver Flt
      OUT     Y0B0  ; Roll    Conv'Fwd
      OUT     T106 K20  ; Roll    Conv'FwdTm
532   LD      B0B1  ; Roll    Conv'RevSw
      OR      X3C9  ; RollConvRev Sw
      ANI     B0B2  ; Roll    Conv'   Stop Sw
      AND     B0E51  ; Manual  ModeLampRoller
      AND     X72  ; Roll    ConveyorOverload
      ANI     Y0B0  ; Roll    Conv'Fwd
      ANI     M6180  ; RollFormConveyorFault
      OUT     Y0B1  ; Roll    Conv'Rev
540   LD      Y0B0  ; Roll    Conv'Fwd
      AND     SM401  ; Normal  Off
      OR      Y0B1  ; Roll    Conv'Rev
      OUT     Y0B2  ; Roll    Conv'   Slow
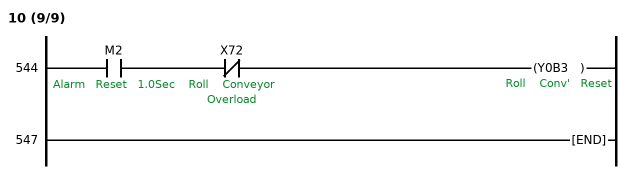
544   LD      M2  ; Alarm   Reset   1.0Sec
      ANI     X72  ; Roll    ConveyorOverload
      OUT     Y0B3  ; Roll    Conv'   Reset
547   END
END_PROGRAM

PROGRAM 100  // #1 Conveyor Part
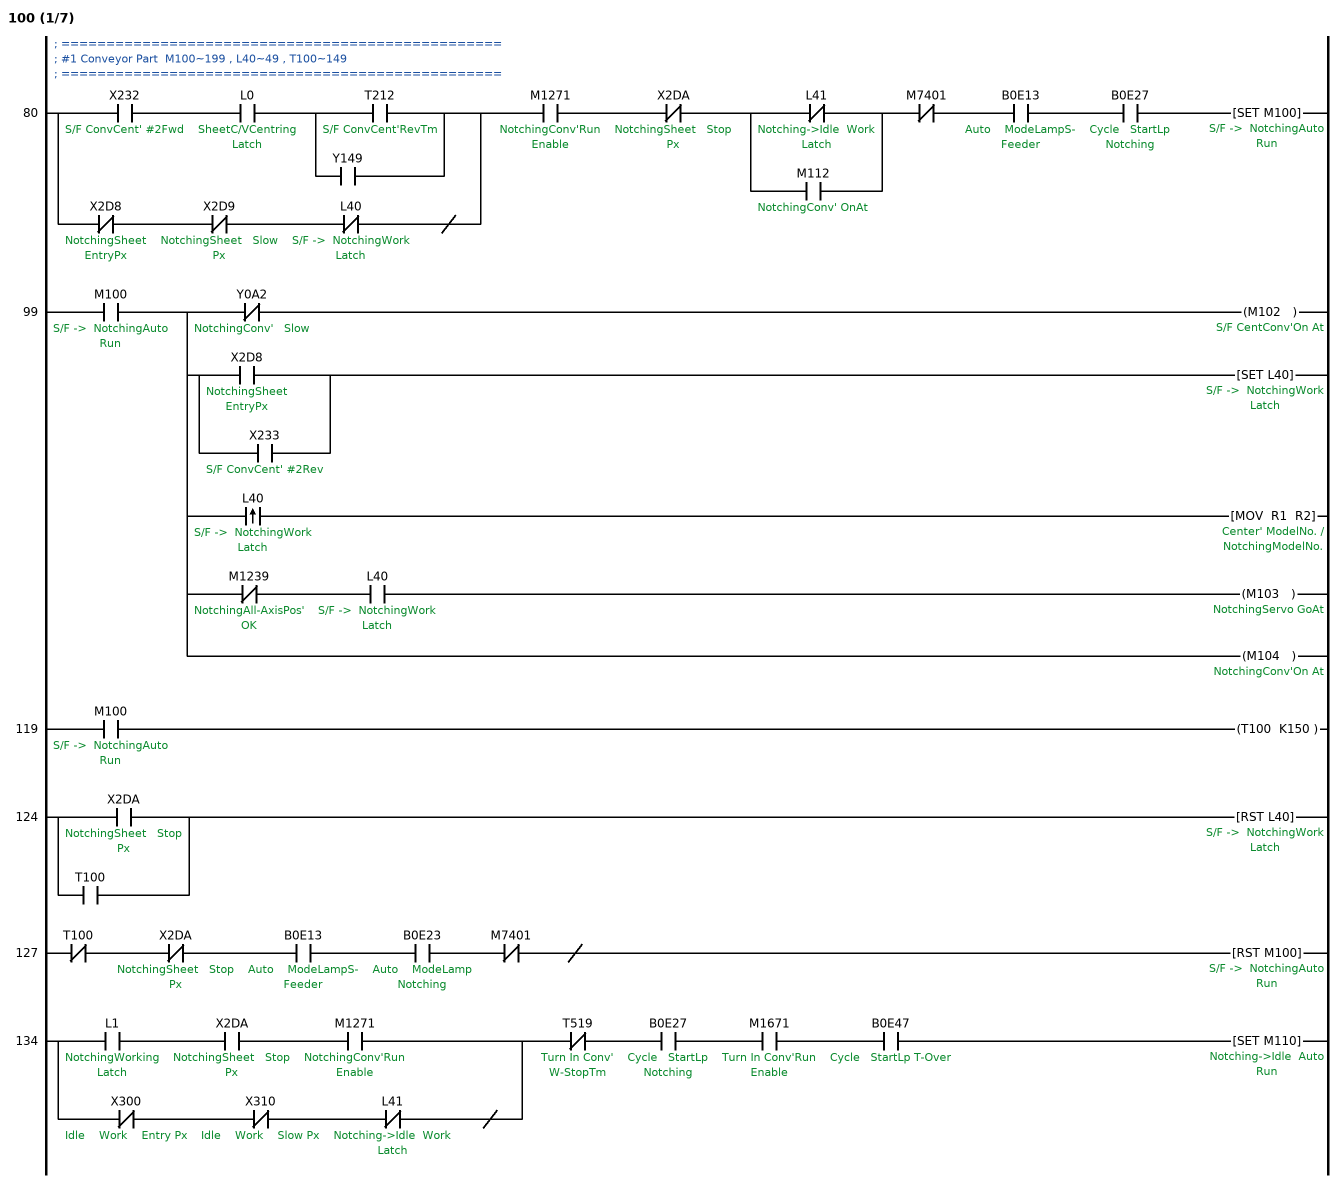
; =================================================
; #1 Conveyor Part  M100~199 , L40~49 , T100~149
; =================================================
80    LD      X232  ; S/F ConvCent' #2Fwd
      AND     L0  ; SheetC/VCentringLatch
      LD      T212  ; S/F ConvCent'RevTm
      OR      Y149
      ANB
      LDI     X2D8  ; NotchingSheet   EntryPx
      ANI     X2D9  ; NotchingSheet   Slow Px
      ANI     L40  ; S/F ->  NotchingWork    Latch
      INV
      ORB
      AND     M1271  ; NotchingConv'RunEnable
      ANI     X2DA  ; NotchingSheet   Stop Px
      LDI     L41  ; Notching->Idle  Work    Latch
      OR      M112  ; NotchingConv' OnAt
      ANB
      ANI     M7401
      AND     B0E13  ; Auto    ModeLampS-Feeder
      AND     B0E27  ; Cycle   StartLp Notching
      SET     M100  ; S/F ->  NotchingAuto Run
99    LD      M100  ; S/F ->  NotchingAuto Run
      MPS
      ANI     Y0A2  ; NotchingConv'   Slow
      OUT     M102  ; S/F CentConv'On At
      MRD
      LD      X2D8  ; NotchingSheet   EntryPx
      OR      X233  ; S/F ConvCent' #2Rev
      ANB
      SET     L40  ; S/F ->  NotchingWork    Latch
      MRD
      ANDP    L40  ; S/F ->  NotchingWork    Latch
      MOV     R1 R2  ; Center' ModelNo. / NotchingModelNo.
      MRD
      ANI     M1239  ; NotchingAll-AxisPos' OK
      AND     L40  ; S/F ->  NotchingWork    Latch
      OUT     M103  ; NotchingServo GoAt
      MPP
      OUT     M104  ; NotchingConv'On At
119   LD      M100  ; S/F ->  NotchingAuto Run
      OUT     T100 K150
124   LD      X2DA  ; NotchingSheet   Stop Px
      OR      T100
      RST     L40  ; S/F ->  NotchingWork    Latch
127   LDI     T100
      ANI     X2DA  ; NotchingSheet   Stop Px
      AND     B0E13  ; Auto    ModeLampS-Feeder
      AND     B0E23  ; Auto    ModeLampNotching
      ANI     M7401
      INV
      RST     M100  ; S/F ->  NotchingAuto Run
134   LD      L1  ; NotchingWorking Latch
      AND     X2DA  ; NotchingSheet   Stop Px
      AND     M1271  ; NotchingConv'RunEnable
      LDI     X300  ; Idle    Work    Entry Px
      ANI     X310  ; Idle    Work    Slow Px
      ANI     L41  ; Notching->Idle  Work    Latch
      INV
      ORB
      ANI     T519  ; Turn In Conv'   W-StopTm
      AND     B0E27  ; Cycle   StartLp Notching
      AND     M1671  ; Turn In Conv'RunEnable
      AND     B0E47  ; Cycle   StartLp T-Over
      SET     M110  ; Notching->Idle  Auto Run
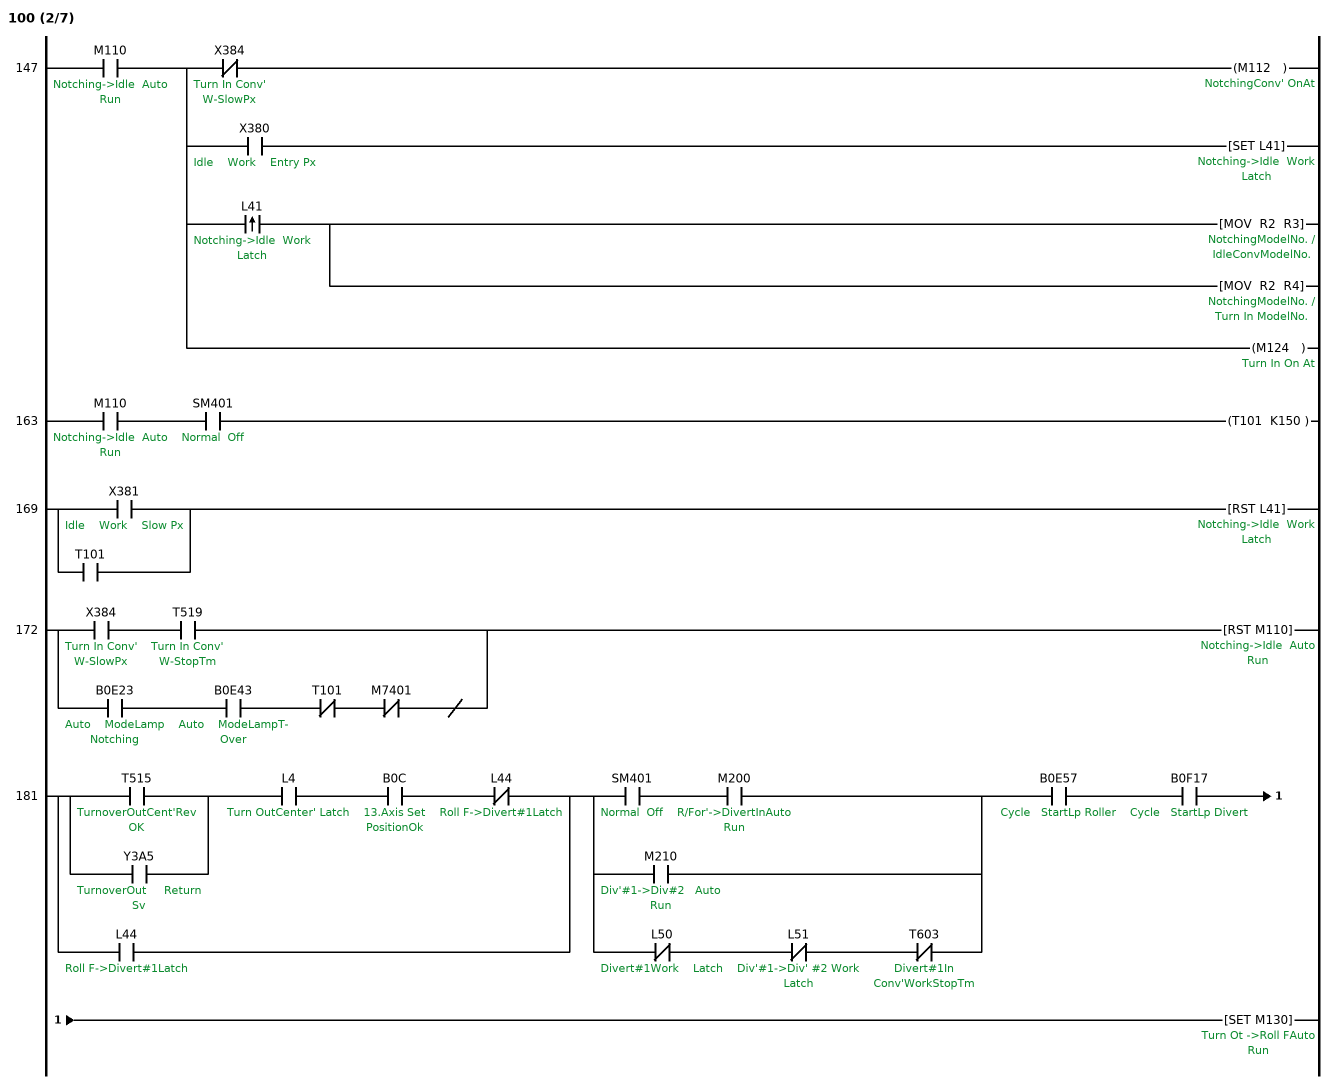
147   LD      M110  ; Notching->Idle  Auto Run
      MPS
      ANI     X384  ; Turn In Conv'   W-SlowPx
      OUT     M112  ; NotchingConv' OnAt
      MRD
      AND     X380  ; Idle    Work    Entry Px
      SET     L41  ; Notching->Idle  Work    Latch
      MRD
      ANDP    L41  ; Notching->Idle  Work    Latch
      MOV     R2 R3  ; IdleConvModelNo.
      MOV     R2 R4  ; Turn In ModelNo.
      MPP
      OUT     M124  ; Turn In On At
163   LD      M110  ; Notching->Idle  Auto Run
      AND     SM401  ; Normal  Off
      OUT     T101 K150
169   LD      X381  ; Idle    Work    Slow Px
      OR      T101
      RST     L41  ; Notching->Idle  Work    Latch
172   LD      X384  ; Turn In Conv'   W-SlowPx
      AND     T519  ; Turn In Conv'   W-StopTm
      LD      B0E23  ; Auto    ModeLampNotching
      AND     B0E43  ; Auto    ModeLampT-Over
      ANI     T101
      ANI     M7401
      INV
      ORB
      RST     M110  ; Notching->Idle  Auto Run
181   LD      T515  ; TurnoverOutCent'Rev OK
      OR      Y3A5  ; TurnoverOut     Return  Sv
      AND     L4  ; Turn OutCenter' Latch
      AND     B0C  ; 13.Axis Set     PositionOk
      ANI     L44  ; Roll F->Divert#1Latch
      OR      L44  ; Roll F->Divert#1Latch
      LD      SM401  ; Normal  Off
      AND     M200  ; R/For'->DivertInAuto Run
      OR      M210  ; Div'#1->Div#2   Auto Run
      LDI     L50  ; Divert#1Work    Latch
      ANI     L51  ; Div'#1->Div' #2 Work    Latch
      ANI     T603  ; Divert#1In Conv'WorkStopTm
      ORB
      ANB
      AND     B0E57  ; Cycle   StartLp Roller
      AND     B0F17  ; Cycle   StartLp Divert
      SET     M130  ; Turn Ot ->Roll FAuto Run
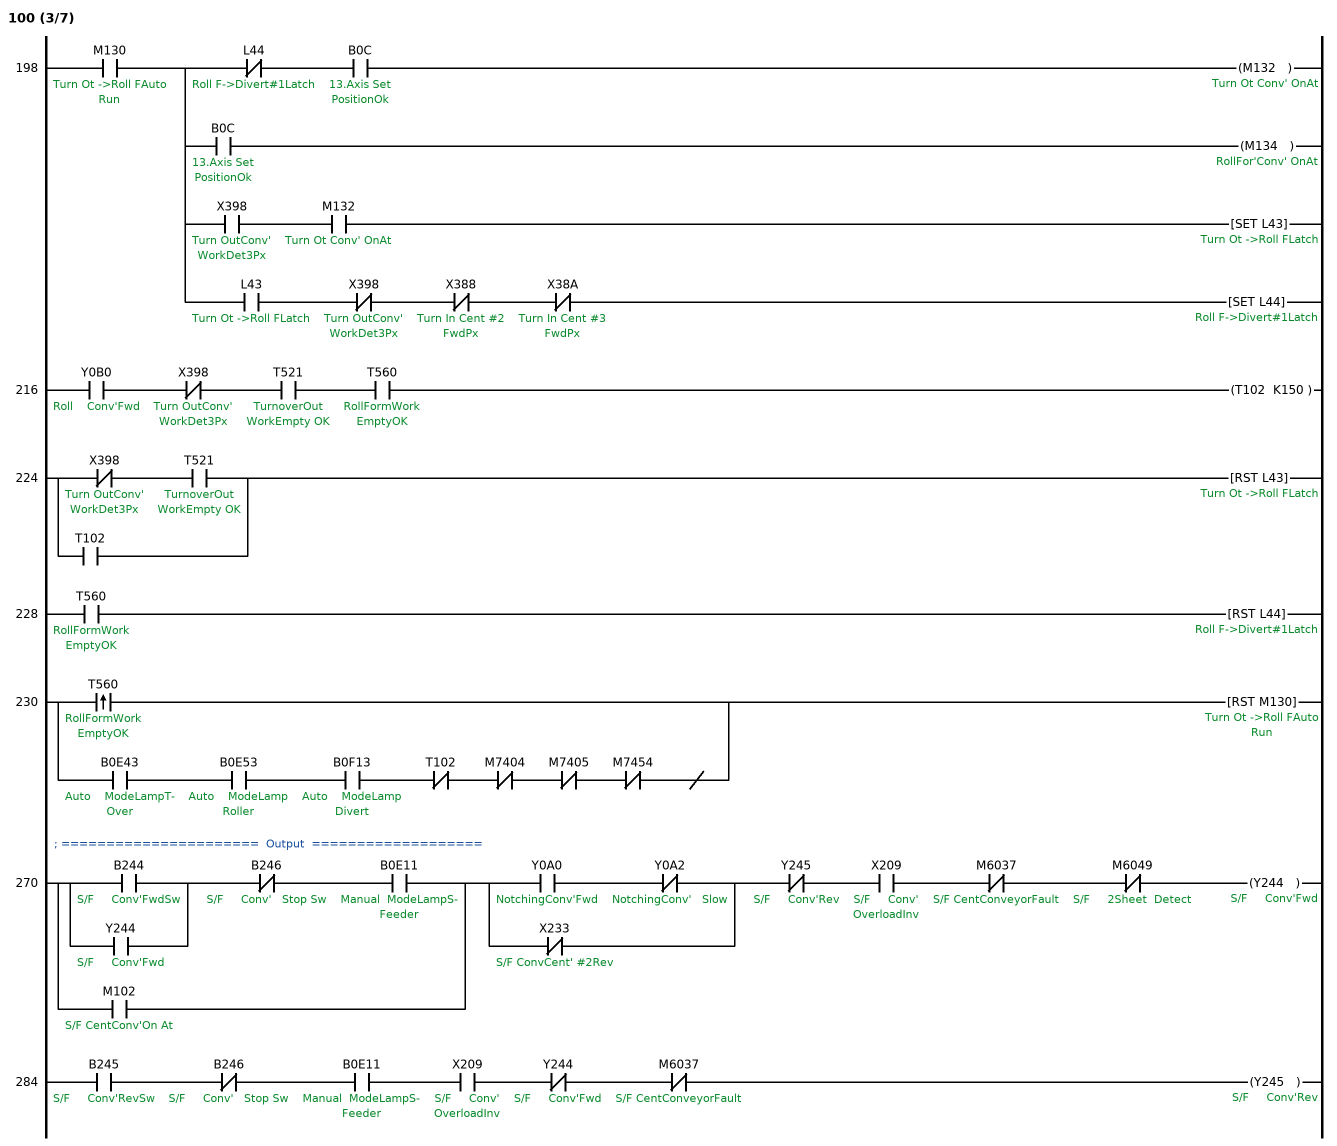
198   LD      M130  ; Turn Ot ->Roll FAuto Run
      MPS
      ANI     L44  ; Roll F->Divert#1Latch
      AND     B0C  ; 13.Axis Set     PositionOk
      OUT     M132  ; Turn Ot Conv' OnAt
      MRD
      AND     B0C  ; 13.Axis Set     PositionOk
      OUT     M134  ; RollFor'Conv' OnAt
      MRD
      AND     X398  ; Turn OutConv'   WorkDet3Px
      AND     M132  ; Turn Ot Conv' OnAt
      SET     L43  ; Turn Ot ->Roll FLatch
      MPP
      AND     L43  ; Turn Ot ->Roll FLatch
      ANI     X398  ; Turn OutConv'   WorkDet3Px
      ANI     X388  ; Turn In Cent #2 FwdPx
      ANI     X38A  ; Turn In Cent #3 FwdPx
      SET     L44  ; Roll F->Divert#1Latch
216   LD      Y0B0  ; Roll    Conv'Fwd
      ANI     X398  ; Turn OutConv'   WorkDet3Px
      AND     T521  ; TurnoverOut WorkEmpty OK
      AND     T560  ; RollFormWork    EmptyOK
      OUT     T102 K150
224   LDI     X398  ; Turn OutConv'   WorkDet3Px
      AND     T521  ; TurnoverOut WorkEmpty OK
      OR      T102
      RST     L43  ; Turn Ot ->Roll FLatch
228   LD      T560  ; RollFormWork    EmptyOK
      RST     L44  ; Roll F->Divert#1Latch
230   LDP     T560  ; RollFormWork    EmptyOK
      LD      B0E43  ; Auto    ModeLampT-Over
      AND     B0E53  ; Auto    ModeLampRoller
      AND     B0F13  ; Auto    ModeLampDivert
      ANI     T102
      ANI     M7404
      ANI     M7405
      ANI     M7454
      INV
      ORB
      RST     M130  ; Turn Ot ->Roll FAuto Run
; ======================  Output  ===================
270   LD      B244  ; S/F     Conv'FwdSw
      OR      Y244  ; S/F     Conv'Fwd
      ANI     B246  ; S/F     Conv'   Stop Sw
      AND     B0E11  ; Manual  ModeLampS-Feeder
      OR      M102  ; S/F CentConv'On At
      LD      Y0A0  ; NotchingConv'Fwd
      ANI     Y0A2  ; NotchingConv'   Slow
      ORI     X233  ; S/F ConvCent' #2Rev
      ANB
      ANI     Y245  ; S/F     Conv'Rev
      AND     X209  ; S/F     Conv'   OverloadInv
      ANI     M6037  ; S/F CentConveyorFault
      ANI     M6049  ; S/F     2Sheet  Detect
      OUT     Y244  ; S/F     Conv'Fwd
284   LD      B245  ; S/F     Conv'RevSw
      ANI     B246  ; S/F     Conv'   Stop Sw
      AND     B0E11  ; Manual  ModeLampS-Feeder
      AND     X209  ; S/F     Conv'   OverloadInv
      ANI     Y244  ; S/F     Conv'Fwd
      ANI     M6037  ; S/F CentConveyorFault
      OUT     Y245  ; S/F     Conv'Rev
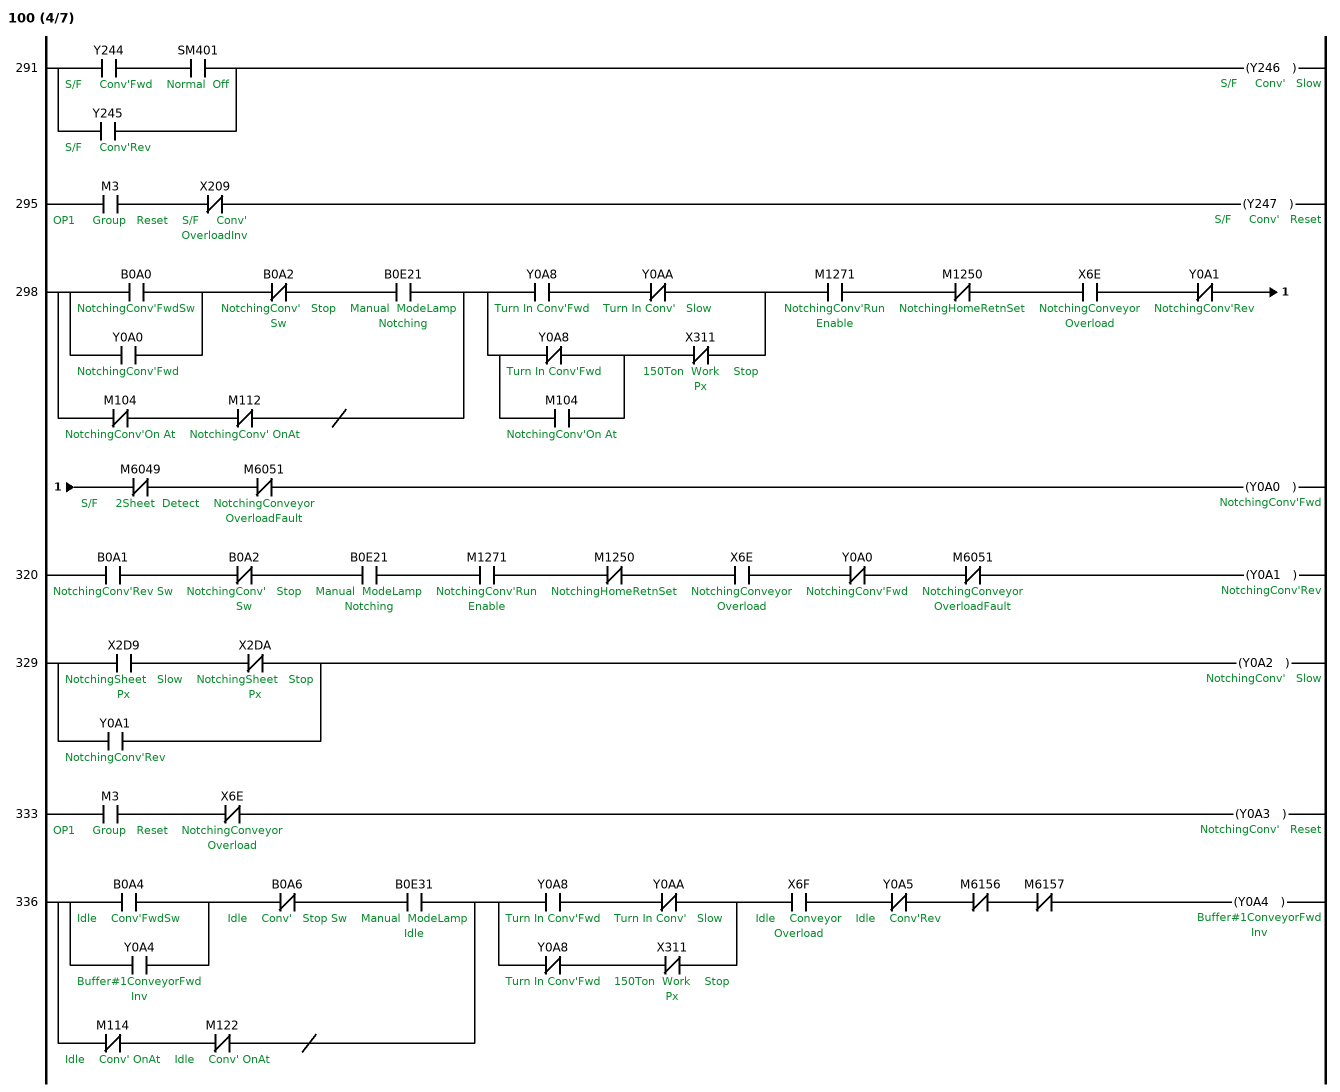
291   LD      Y244  ; S/F     Conv'Fwd
      AND     SM401  ; Normal  Off
      OR      Y245  ; S/F     Conv'Rev
      OUT     Y246  ; S/F     Conv'   Slow
295   LD      M3  ; OP1     Group   Reset
      ANI     X209  ; S/F     Conv'   OverloadInv
      OUT     Y247  ; S/F     Conv'   Reset
298   LD      B0A0  ; NotchingConv'FwdSw
      OR      Y0A0  ; NotchingConv'Fwd
      ANI     B0A2  ; NotchingConv'   Stop Sw
      AND     B0E21  ; Manual  ModeLampNotching
      LDI     M104  ; NotchingConv'On At
      ANI     M112  ; NotchingConv' OnAt
      INV
      ORB
      LD      Y0A8  ; Turn In Conv'Fwd
      ANI     Y0AA  ; Turn In Conv'   Slow
      LDI     Y0A8  ; Turn In Conv'Fwd
      OR      M104  ; NotchingConv'On At
      ANI     X311  ; 150Ton  Work    Stop Px
      ORB
      ANB
      AND     M1271  ; NotchingConv'RunEnable
      ANI     M1250  ; NotchingHomeRetnSet
      AND     X6E  ; NotchingConveyorOverload
      ANI     Y0A1  ; NotchingConv'Rev
      ANI     M6049  ; S/F     2Sheet  Detect
      ANI     M6051  ; NotchingConveyorOverloadFault
      OUT     Y0A0  ; NotchingConv'Fwd
320   LD      B0A1  ; NotchingConv'Rev Sw
      ANI     B0A2  ; NotchingConv'   Stop Sw
      AND     B0E21  ; Manual  ModeLampNotching
      AND     M1271  ; NotchingConv'RunEnable
      ANI     M1250  ; NotchingHomeRetnSet
      AND     X6E  ; NotchingConveyorOverload
      ANI     Y0A0  ; NotchingConv'Fwd
      ANI     M6051  ; NotchingConveyorOverloadFault
      OUT     Y0A1  ; NotchingConv'Rev
329   LD      X2D9  ; NotchingSheet   Slow Px
      ANI     X2DA  ; NotchingSheet   Stop Px
      OR      Y0A1  ; NotchingConv'Rev
      OUT     Y0A2  ; NotchingConv'   Slow
333   LD      M3  ; OP1     Group   Reset
      ANI     X6E  ; NotchingConveyorOverload
      OUT     Y0A3  ; NotchingConv'   Reset
336   LD      B0A4  ; Idle    Conv'FwdSw
      OR      Y0A4  ; Buffer#1ConveyorFwd Inv
      ANI     B0A6  ; Idle    Conv'   Stop Sw
      AND     B0E31  ; Manual  ModeLampIdle
      LDI     M114  ; Idle    Conv' OnAt
      ANI     M122  ; Idle    Conv' OnAt
      INV
      ORB
      LD      Y0A8  ; Turn In Conv'Fwd
      ANI     Y0AA  ; Turn In Conv'   Slow
      LDI     Y0A8  ; Turn In Conv'Fwd
      ANI     X311  ; 150Ton  Work    Stop Px
      ORB
      ANB
      AND     X6F  ; Idle    ConveyorOverload
      ANI     Y0A5  ; Idle    Conv'Rev
      ANI     M6156
      ANI     M6157
      OUT     Y0A4  ; Buffer#1ConveyorFwd Inv
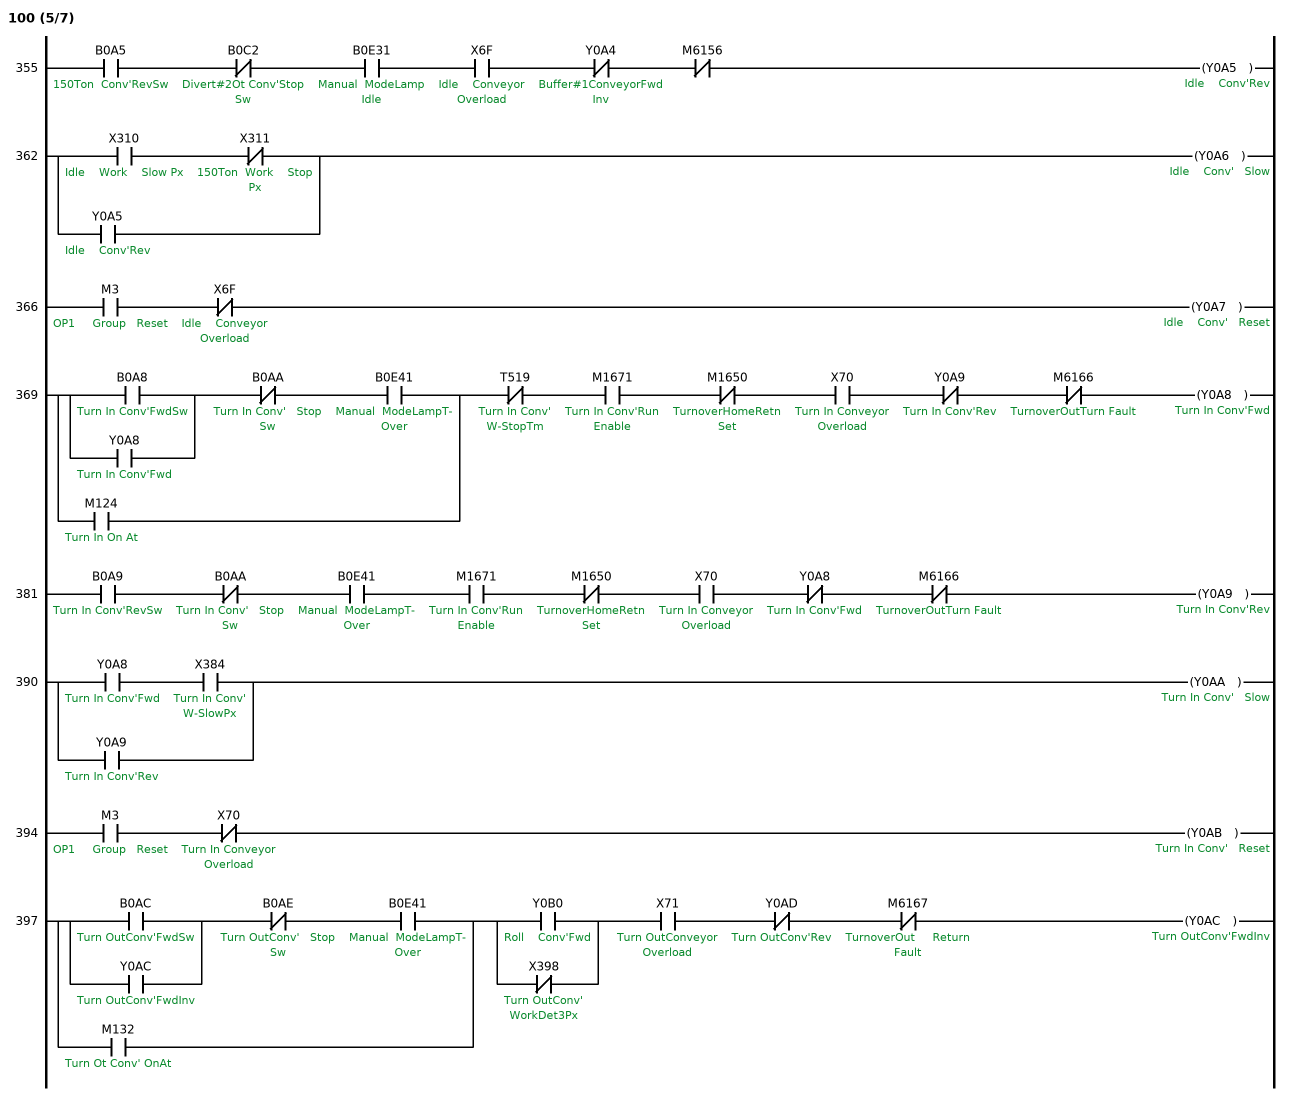
355   LD      B0A5  ; 150Ton  Conv'RevSw
      ANI     B0C2  ; Divert#2Ot Conv'Stop Sw
      AND     B0E31  ; Manual  ModeLampIdle
      AND     X6F  ; Idle    ConveyorOverload
      ANI     Y0A4  ; Buffer#1ConveyorFwd Inv
      ANI     M6156
      OUT     Y0A5  ; Idle    Conv'Rev
362   LD      X310  ; Idle    Work    Slow Px
      ANI     X311  ; 150Ton  Work    Stop Px
      OR      Y0A5  ; Idle    Conv'Rev
      OUT     Y0A6  ; Idle    Conv'   Slow
366   LD      M3  ; OP1     Group   Reset
      ANI     X6F  ; Idle    ConveyorOverload
      OUT     Y0A7  ; Idle    Conv'   Reset
369   LD      B0A8  ; Turn In Conv'FwdSw
      OR      Y0A8  ; Turn In Conv'Fwd
      ANI     B0AA  ; Turn In Conv'   Stop Sw
      AND     B0E41  ; Manual  ModeLampT-Over
      OR      M124  ; Turn In On At
      ANI     T519  ; Turn In Conv'   W-StopTm
      AND     M1671  ; Turn In Conv'RunEnable
      ANI     M1650  ; TurnoverHomeRetnSet
      AND     X70  ; Turn In ConveyorOverload
      ANI     Y0A9  ; Turn In Conv'Rev
      ANI     M6166  ; TurnoverOutTurn Fault
      OUT     Y0A8  ; Turn In Conv'Fwd
381   LD      B0A9  ; Turn In Conv'RevSw
      ANI     B0AA  ; Turn In Conv'   Stop Sw
      AND     B0E41  ; Manual  ModeLampT-Over
      AND     M1671  ; Turn In Conv'RunEnable
      ANI     M1650  ; TurnoverHomeRetnSet
      AND     X70  ; Turn In ConveyorOverload
      ANI     Y0A8  ; Turn In Conv'Fwd
      ANI     M6166  ; TurnoverOutTurn Fault
      OUT     Y0A9  ; Turn In Conv'Rev
390   LD      Y0A8  ; Turn In Conv'Fwd
      AND     X384  ; Turn In Conv'   W-SlowPx
      OR      Y0A9  ; Turn In Conv'Rev
      OUT     Y0AA  ; Turn In Conv'   Slow
394   LD      M3  ; OP1     Group   Reset
      ANI     X70  ; Turn In ConveyorOverload
      OUT     Y0AB  ; Turn In Conv'   Reset
397   LD      B0AC  ; Turn OutConv'FwdSw
      OR      Y0AC  ; Turn OutConv'FwdInv
      ANI     B0AE  ; Turn OutConv'   Stop Sw
      AND     B0E41  ; Manual  ModeLampT-Over
      OR      M132  ; Turn Ot Conv' OnAt
      LD      Y0B0  ; Roll    Conv'Fwd
      ORI     X398  ; Turn OutConv'   WorkDet3Px
      ANB
      AND     X71  ; Turn OutConveyorOverload
      ANI     Y0AD  ; Turn OutConv'Rev
      ANI     M6167  ; TurnoverOut     Return  Fault
      OUT     Y0AC  ; Turn OutConv'FwdInv
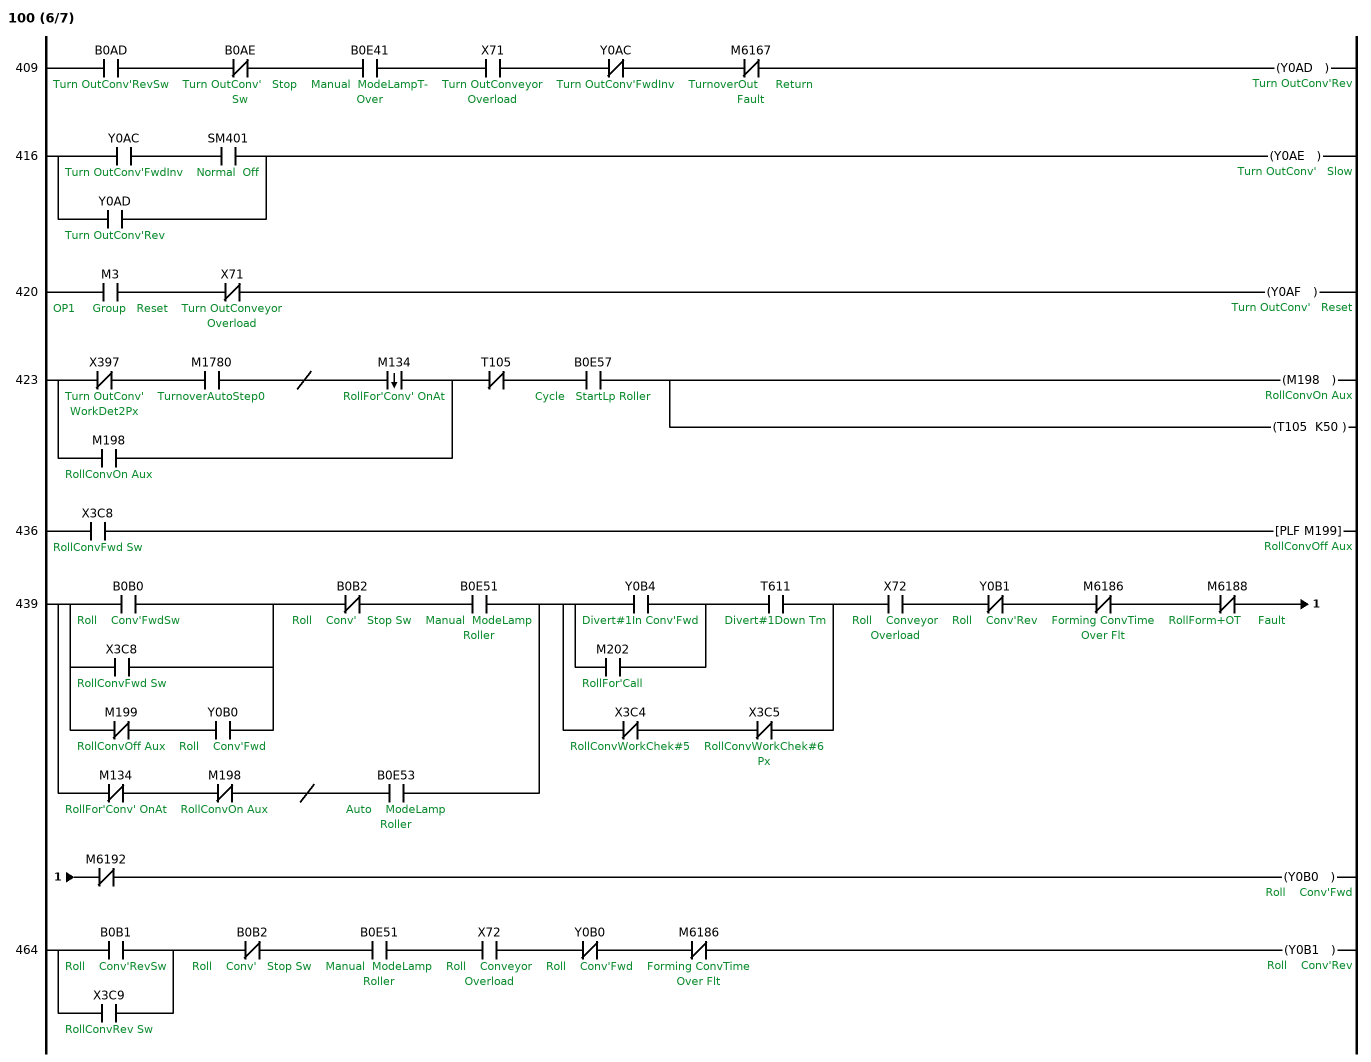
409   LD      B0AD  ; Turn OutConv'RevSw
      ANI     B0AE  ; Turn OutConv'   Stop Sw
      AND     B0E41  ; Manual  ModeLampT-Over
      AND     X71  ; Turn OutConveyorOverload
      ANI     Y0AC  ; Turn OutConv'FwdInv
      ANI     M6167  ; TurnoverOut     Return  Fault
      OUT     Y0AD  ; Turn OutConv'Rev
416   LD      Y0AC  ; Turn OutConv'FwdInv
      AND     SM401  ; Normal  Off
      OR      Y0AD  ; Turn OutConv'Rev
      OUT     Y0AE  ; Turn OutConv'   Slow
420   LD      M3  ; OP1     Group   Reset
      ANI     X71  ; Turn OutConveyorOverload
      OUT     Y0AF  ; Turn OutConv'   Reset
423   LDI     X397  ; Turn OutConv'   WorkDet2Px
      AND     M1780  ; TurnoverAutoStep0
      INV
      ANDF    M134  ; RollFor'Conv' OnAt
      OR      M198  ; RollConvOn Aux
      ANI     T105
      AND     B0E57  ; Cycle   StartLp Roller
      OUT     M198  ; RollConvOn Aux
      OUT     T105 K50
436   LD      X3C8  ; RollConvFwd Sw
      PLF     M199  ; RollConvOff Aux
439   LD      B0B0  ; Roll    Conv'FwdSw
      OR      X3C8  ; RollConvFwd Sw
      LDI     M199  ; RollConvOff Aux
      AND     Y0B0  ; Roll    Conv'Fwd
      ORB
      ANI     B0B2  ; Roll    Conv'   Stop Sw
      AND     B0E51  ; Manual  ModeLampRoller
      LDI     M134  ; RollFor'Conv' OnAt
      ANI     M198  ; RollConvOn Aux
      INV
      AND     B0E53  ; Auto    ModeLampRoller
      ORB
      LD      Y0B4  ; Divert#1In Conv'Fwd
      OR      M202  ; RollFor'Call
      AND     T611  ; Divert#1Down Tm
      LDI     X3C4  ; RollConvWorkChek#5
      ANI     X3C5  ; RollConvWorkChek#6 Px
      ORB
      ANB
      AND     X72  ; Roll    ConveyorOverload
      ANI     Y0B1  ; Roll    Conv'Rev
      ANI     M6186  ; Forming ConvTimeOver Flt
      ANI     M6188  ; RollForm+OT     Fault
      ANI     M6192
      OUT     Y0B0  ; Roll    Conv'Fwd
464   LD      B0B1  ; Roll    Conv'RevSw
      OR      X3C9  ; RollConvRev Sw
      ANI     B0B2  ; Roll    Conv'   Stop Sw
      AND     B0E51  ; Manual  ModeLampRoller
      AND     X72  ; Roll    ConveyorOverload
      ANI     Y0B0  ; Roll    Conv'Fwd
      ANI     M6186  ; Forming ConvTimeOver Flt
      OUT     Y0B1  ; Roll    Conv'Rev
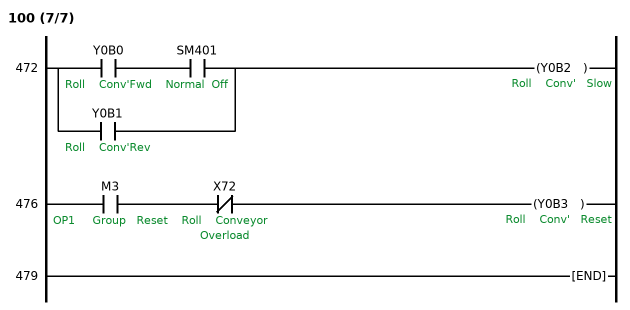
472   LD      Y0B0  ; Roll    Conv'Fwd
      AND     SM401  ; Normal  Off
      OR      Y0B1  ; Roll    Conv'Rev
      OUT     Y0B2  ; Roll    Conv'   Slow
476   LD      M3  ; OP1     Group   Reset
      ANI     X72  ; Roll    ConveyorOverload
      OUT     Y0B3  ; Roll    Conv'   Reset
479   END
END_PROGRAM

PROGRAM 11  // Sheet Feed
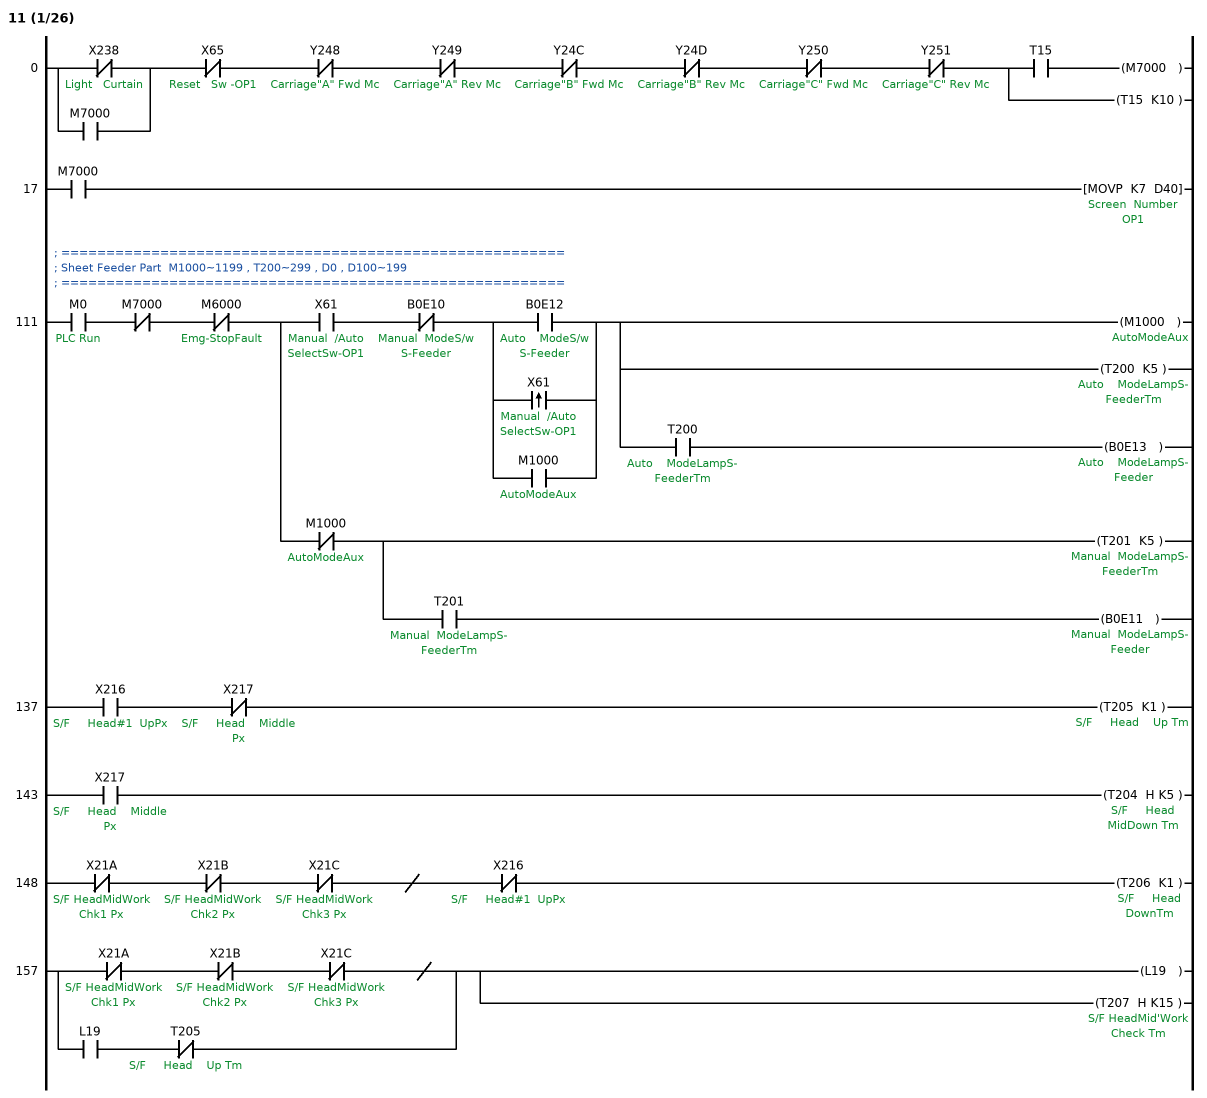
0     LDI     X238  ; Light   Curtain
      OR      M7000
      ANI     X65  ; Reset   Sw -OP1
      ANI     Y248  ; Carriage"A" Fwd Mc
      ANI     Y249  ; Carriage"A" Rev Mc
      ANI     Y24C  ; Carriage"B" Fwd Mc
      ANI     Y24D  ; Carriage"B" Rev Mc
      ANI     Y250  ; Carriage"C" Fwd Mc
      ANI     Y251  ; Carriage"C" Rev Mc
      MPS
      AND     T15
      OUT     M7000
      MPP
      OUT     T15 K10
17    LD      M7000
      MOVP    K7 D40  ; Screen  Number  OP1
; ========================================================
; Sheet Feeder Part  M1000~1199 , T200~299 , D0 , D100~199
; ========================================================
111   LD      M0  ; PLC Run
      ANI     M7000
      ANI     M6000  ; Emg-StopFault
      MPS
      AND     X61  ; Manual  /Auto   SelectSw-OP1
      ANI     B0E10  ; Manual  ModeS/w S-Feeder
      LD      B0E12  ; Auto    ModeS/w S-Feeder
      ORP     X61  ; Manual  /Auto   SelectSw-OP1
      OR      M1000  ; AutoModeAux
      ANB
      OUT     M1000  ; AutoModeAux
      OUT     T200 K5  ; Auto    ModeLampS-FeederTm
      AND     T200  ; Auto    ModeLampS-FeederTm
      OUT     B0E13  ; Auto    ModeLampS-Feeder
      MPP
      ANI     M1000  ; AutoModeAux
      OUT     T201 K5  ; Manual  ModeLampS-FeederTm
      AND     T201  ; Manual  ModeLampS-FeederTm
      OUT     B0E11  ; Manual  ModeLampS-Feeder
137   LD      X216  ; S/F     Head#1  UpPx
      ANI     X217  ; S/F     Head    Middle  Px
      OUT     T205 K1  ; S/F     Head    Up Tm
143   LD      X217  ; S/F     Head    Middle  Px
      OUTH    T204 K5  ; S/F     Head    MidDown Tm
148   LDI     X21A  ; S/F HeadMidWork Chk1 Px
      ANI     X21B  ; S/F HeadMidWork Chk2 Px
      ANI     X21C  ; S/F HeadMidWork Chk3 Px
      INV
      ANI     X216  ; S/F     Head#1  UpPx
      OUT     T206 K1  ; S/F     Head    DownTm
157   LDI     X21A  ; S/F HeadMidWork Chk1 Px
      ANI     X21B  ; S/F HeadMidWork Chk2 Px
      ANI     X21C  ; S/F HeadMidWork Chk3 Px
      INV
      LD      L19
      ANI     T205  ; S/F     Head    Up Tm
      ORB
      OUT     L19
      OUTH    T207 K15  ; S/F HeadMid'WorkCheck Tm
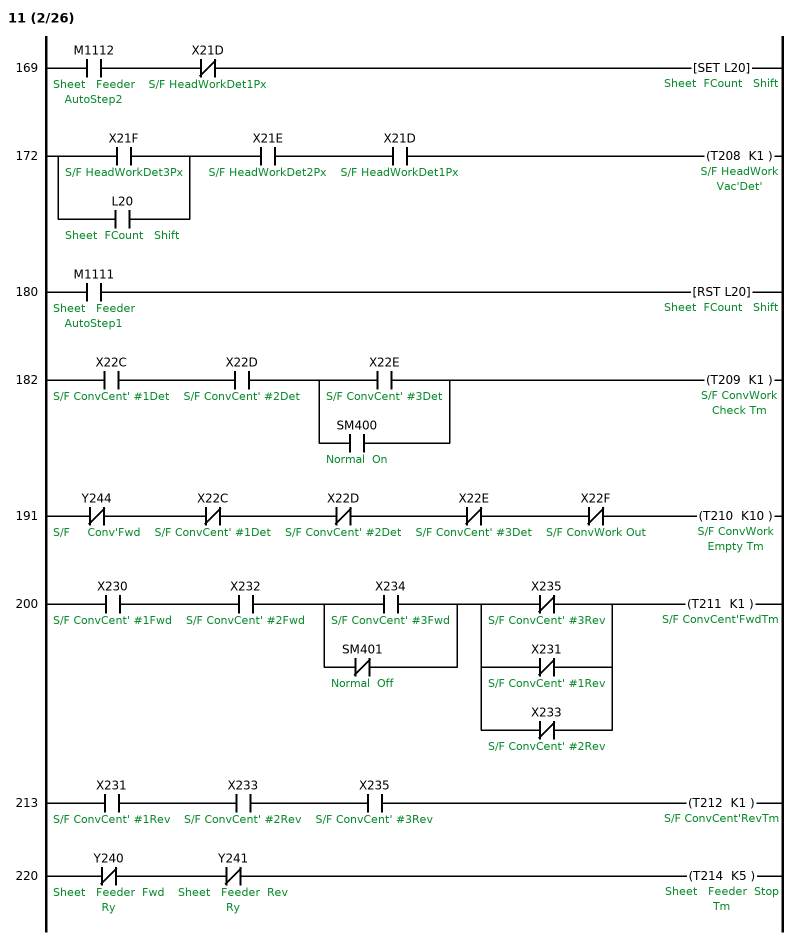
169   LD      M1112  ; Sheet   Feeder  AutoStep2
      ANI     X21D  ; S/F HeadWorkDet1Px
      SET     L20  ; Sheet  FCount   Shift
172   LD      X21F  ; S/F HeadWorkDet3Px
      OR      L20  ; Sheet  FCount   Shift
      AND     X21E  ; S/F HeadWorkDet2Px
      AND     X21D  ; S/F HeadWorkDet1Px
      OUT     T208 K1  ; S/F HeadWorkVac'Det'
180   LD      M1111  ; Sheet   Feeder  AutoStep1
      RST     L20  ; Sheet  FCount   Shift
182   LD      X22C  ; S/F ConvCent' #1Det
      AND     X22D  ; S/F ConvCent' #2Det
      LD      X22E  ; S/F ConvCent' #3Det
      OR      SM400  ; Normal  On
      ANB
      OUT     T209 K1  ; S/F ConvWork    Check Tm
191   LDI     Y244  ; S/F     Conv'Fwd
      ANI     X22C  ; S/F ConvCent' #1Det
      ANI     X22D  ; S/F ConvCent' #2Det
      ANI     X22E  ; S/F ConvCent' #3Det
      ANI     X22F  ; S/F ConvWork Out
      OUT     T210 K10  ; S/F ConvWork    Empty Tm
200   LD      X230  ; S/F ConvCent' #1Fwd
      AND     X232  ; S/F ConvCent' #2Fwd
      LD      X234  ; S/F ConvCent' #3Fwd
      ORI     SM401  ; Normal  Off
      ANB
      LDI     X235  ; S/F ConvCent' #3Rev
      ORI     X231  ; S/F ConvCent' #1Rev
      ORI     X233  ; S/F ConvCent' #2Rev
      ANB
      OUT     T211 K1  ; S/F ConvCent'FwdTm
213   LD      X231  ; S/F ConvCent' #1Rev
      AND     X233  ; S/F ConvCent' #2Rev
      AND     X235  ; S/F ConvCent' #3Rev
      OUT     T212 K1  ; S/F ConvCent'RevTm
220   LDI     Y240  ; Sheet   Feeder  Fwd Ry
      ANI     Y241  ; Sheet   Feeder  Rev Ry
      OUT     T214 K5  ; Sheet   Feeder  Stop Tm
